LIN {X 0,Y 207.19,Z 445.671,A -85,B 0,C 180,E1 -21067.798,E2 -21067.798} C_VEL
LIN {X 0,Y 206.976,Z 445.696,A -85,B 0,C 180,E1 -21071.756,E2 -21071.756} C_VEL
LIN {X 0,Y 206.869,Z 445.715,A -85,B 0,C 180,E1 -21075.771,E2 -21075.771} C_VEL
LIN {X 0,Y 206.785,Z 445.706,A -85,B 0,C 180,E1 -21079.869,E2 -21079.869} C_VEL
LIN {X 0,Y 206.765,Z 445.704,A -85,B 0,C 180,E1 -21084.072,E2 -21084.072} C_VEL
LIN {X 0,Y 206.745,Z 445.731,A -85,B 0,C 180,E1 -21088.419,E2 -21088.419} C_VEL
LIN {X 0,Y 206.71,Z 445.707,A -85,B 0,C 180,E1 -21092.956,E2 -21092.956} C_VEL
LIN {X 0,Y 206.723,Z 445.722,A -85,B 0,C 180,E1 -21095.321,E2 -21095.321} C_VEL
LIN {X 0,Y 206.668,Z 445.735,A -85,B 0,C 180,E1 -21100.25,E2 -21100.25} C_VEL
LIN {X 0,Y 206.636,Z 445.739,A -85,B 0,C 180,E1 -21105.582,E2 -21105.582} C_VEL
LIN {X 0,Y 206.668,Z 445.737,A -85,B 0,C 180,E1 -21109.751,E2 -21109.751} C_VEL
LIN {X 0,Y 206.733,Z 445.724,A -85,B 0,C 180,E1 -21114.696,E2 -21114.696} C_VEL
LIN {X 0,Y 206.73,Z 445.73,A -85,B 0,C 180,E1 -21119.52,E2 -21119.52} C_VEL
LIN {X 0,Y 207.05,Z 447.125,A -85,B 0,C 180,E1 -21119.722,E2 -21119.722} C_VEL
LIN {X 0,Y 211.426,Z 456.277,A -85,B 0,C 180,E1 -21121.603,E2 -21121.603} C_VEL
LIN {X 0,Y 214.653,Z 464.205,A -85,B 0,C 180,E1 -21123.308,E2 -21123.308} C_VEL
LIN {X 0,Y 217.835,Z 474.221,A -85,B 0,C 180,E1 -21125.577,E2 -21125.577} C_VEL
LIN {X 0,Y 220.061,Z 483.327,A -85,B 0,C 180,E1 -21127.846,E2 -21127.846} C_VEL
LIN {X 0,Y 218.248,Z 491.893,A -85,B 0,C 180,E1 -21129.747,E2 -21129.747} C_VEL
LIN {X 0,Y 215.992,Z 500.319,A -85,B 0,C 180,E1 -21131.995,E2 -21131.995} C_VEL
LIN {X 0,Y 213.676,Z 508.48,A -85,B 0,C 180,E1 -21134.745,E2 -21134.745} C_VEL
LIN {X 0,Y 211.802,Z 515.035,A -85,B 0,C 180,E1 -21137.545,E2 -21137.545} C_VEL
LIN {X 0,Y 210.29,Z 520.267,A -85,B 0,C 180,E1 -21140.381,E2 -21140.381} C_VEL
LIN {X 0,Y 209.024,Z 524.37,A -85,B 0,C 180,E1 -21143.242,E2 -21143.242} C_VEL
LIN {X 0,Y 207.997,Z 527.462,A -85,B 0,C 180,E1 -21146.126,E2 -21146.126} C_VEL
LIN {X 0,Y 207.633,Z 528.989,A -85,B 0,C 180,E1 -21148.061,E2 -21148.061} C_VEL
LIN {X 0,Y 207.465,Z 530.098,A -85,B 0,C 180,E1 -21150,E2 -21150} C_VEL
LIN {X 0,Y 207.463,Z 530.79,A -85,B 0,C 180,E1 -21151.942,E2 -21151.942} C_VEL
LIN {X 0,Y 207.447,Z 531.134,A -85,B 0,C 180,E1 -21155.834,E2 -21155.834} C_VEL
LIN {X 0,Y 207.905,Z 530.696,A -85,B 0,C 180,E1 -21157.772,E2 -21157.772} C_VEL
LIN {X 0,Y 209.475,Z 528.577,A -85,B 0,C 180,E1 -21161.614,E2 -21161.614} C_VEL
LIN {X 0,Y 211.112,Z 525.293,A -85,B 0,C 180,E1 -21165.109,E2 -21165.109} C_VEL
LIN {X 0,Y 212.98,Z 520.951,A -85,B 0,C 180,E1 -21168.27,E2 -21168.27} C_VEL
LIN {X 0,Y 215.03,Z 515.843,A -85,B 0,C 180,E1 -21171.071,E2 -21171.071} C_VEL
LIN {X 0,Y 217.394,Z 509.41,A -85,B 0,C 180,E1 -21173.836,E2 -21173.836} C_VEL
LIN {X 0,Y 220.287,Z 501.361,A -85,B 0,C 180,E1 -21176.53,E2 -21176.53} C_VEL
LIN {X 0,Y 222.893,Z 493.095,A -85,B 0,C 180,E1 -21178.741,E2 -21178.741} C_VEL
LIN {X 0,Y 223.378,Z 491.199,A -85,B 0,C 180,E1 -21179.188,E2 -21179.188} C_VEL
LIN {X 0,Y 223.029,Z 487.399,A -85,B 0,C 180,E1 -21180.278,E2 -21180.278} C_VEL
LIN {X 0,Y 220.921,Z 478.734,A -85,B 0,C 180,E1 -21182.739,E2 -21182.739} C_VEL
LIN {X 0,Y 217.615,Z 468.861,A -85,B 0,C 180,E1 -21185.368,E2 -21185.368} C_VEL
LIN {X 0,Y 213.924,Z 460.069,A -85,B 0,C 180,E1 -21187.6,E2 -21187.6} C_VEL
LIN {X 0,Y 210.239,Z 452.835,A -85,B 0,C 180,E1 -21189.431,E2 -21189.431} C_VEL
LIN {X 0,Y 208.72,Z 449.857,A -85,B 0,C 180,E1 -21190.156,E2 -21190.156} C_VEL
LIN {X 0,Y 207.001,Z 447.117,A -85,B 0,C 180,E1 -21190.871,E2 -21190.871} C_VEL
LIN {X 0,Y 206.686,Z 445.74,A -85,B 0,C 180,E1 -21191.119,E2 -21191.119} C_VEL
LIN {X 0,Y 206.638,Z 445.745,A -85,B 0,C 180,E1 -21195.581,E2 -21195.581} C_VEL
LIN {X 0,Y 206.67,Z 445.738,A -85,B 0,C 180,E1 -21199.75,E2 -21199.75} C_VEL
LIN {X 0,Y 206.735,Z 445.729,A -85,B 0,C 180,E1 -21204.695,E2 -21204.695} C_VEL
LIN {X 0,Y 206.728,Z 445.732,A -85,B 0,C 180,E1 -21209.339,E2 -21209.339} C_VEL
LIN {X 0,Y 206.735,Z 445.734,A -85,B 0,C 180,E1 -21213.772,E2 -21213.772} C_VEL
LIN {X 0,Y 206.86,Z 445.715,A -85,B 0,C 180,E1 -21219.1,E2 -21219.1} C_VEL
LIN {X 0,Y 206.941,Z 445.761,A -85,B 0,C 180,E1 -21219.693,E2 -21219.693} C_VEL
LIN {X 0,Y 209.859,Z 459.288,A -85,B 0,C 180,E1 -21221.594,E2 -21221.594} C_VEL
LIN {X 0,Y 210.707,Z 463.779,A -85,B 0,C 180,E1 -21222.316,E2 -21222.316} C_VEL
LIN {X 0,Y 209.71,Z 475.714,A -85,B 0,C 180,E1 -21224.448,E2 -21224.448} C_VEL
LIN {X 0,Y 208.543,Z 487.804,A -85,B 0,C 180,E1 -21227.099,E2 -21227.099} C_VEL
LIN {X 0,Y 207.569,Z 498.303,A -85,B 0,C 180,E1 -21229.914,E2 -21229.914} C_VEL
LIN {X 0,Y 206.894,Z 506.907,A -85,B 0,C 180,E1 -21232.681,E2 -21232.681} C_VEL
LIN {X 0,Y 206.491,Z 514.452,A -85,B 0,C 180,E1 -21235.608,E2 -21235.608} C_VEL
LIN {X 0,Y 206.658,Z 521.636,A -85,B 0,C 180,E1 -21239.025,E2 -21239.025} C_VEL
LIN {X 0,Y 207.102,Z 526.662,A -85,B 0,C 180,E1 -21241.944,E2 -21241.944} C_VEL
LIN {X 0,Y 208.248,Z 531.871,A -85,B 0,C 180,E1 -21245.811,E2 -21245.811} C_VEL
LIN {X 0,Y 210.256,Z 535.477,A -85,B 0,C 180,E1 -21249.621,E2 -21249.621} C_VEL
LIN {X 0,Y 213.286,Z 537.641,A -85,B 0,C 180,E1 -21253.336,E2 -21253.336} C_VEL
LIN {X 0,Y 216.951,Z 538.342,A -85,B 0,C 180,E1 -21256.951,E2 -21256.951} C_VEL
LIN {X 0,Y 221.52,Z 537.675,A -85,B 0,C 180,E1 -21260.425,E2 -21260.425} C_VEL
LIN {X 0,Y 226.914,Z 535.59,A -85,B 0,C 180,E1 -21263.743,E2 -21263.743} C_VEL
LIN {X 0,Y 233.04,Z 532.075,A -85,B 0,C 180,E1 -21266.896,E2 -21266.896} C_VEL
LIN {X 0,Y 239.903,Z 527.051,A -85,B 0,C 180,E1 -21269.869,E2 -21269.869} C_VEL
LIN {X 0,Y 247.431,Z 520.392,A -85,B 0,C 180,E1 -21272.661,E2 -21272.661} C_VEL
LIN {X 0,Y 248.551,Z 519.043,A -85,B 0,C 180,E1 -21273.462,E2 -21273.462} C_VEL
LIN {X 0,Y 249.773,Z 517.18,A -85,B 0,C 180,E1 -21275.314,E2 -21275.314} C_VEL
LIN {X 0,Y 250.027,Z 516.636,A -85,B 0,C 180,E1 -21276.177,E2 -21276.177} C_VEL
LIN {X 0,Y 250.154,Z 516.146,A -85,B 0,C 180,E1 -21278.176,E2 -21278.176} C_VEL
LIN {X 0,Y 249.645,Z 516.912,A -85,B 0,C 180,E1 -21280.526,E2 -21280.526} C_VEL
LIN {X 0,Y 248.76,Z 518.828,A -85,B 0,C 180,E1 -21282.73,E2 -21282.73} C_VEL
LIN {X 0,Y 248.092,Z 520.223,A -85,B 0,C 180,E1 -21283.715,E2 -21283.715} C_VEL
LIN {X 0,Y 247.046,Z 522.094,A -85,B 0,C 180,E1 -21284.666,E2 -21284.666} C_VEL
LIN {X 0,Y 243.621,Z 527.852,A -85,B 0,C 180,E1 -21286.954,E2 -21286.954} C_VEL
LIN {X 0,Y 238.302,Z 537.311,A -85,B 0,C 180,E1 -21290.471,E2 -21290.471} C_VEL
LIN {X 0,Y 232.802,Z 546.857,A -85,B 0,C 180,E1 -21293.936,E2 -21293.936} C_VEL
LIN {X 0,Y 227.947,Z 554.484,A -85,B 0,C 180,E1 -21296.82,E2 -21296.82} C_VEL
LIN {X 0,Y 221.36,Z 563.244,A -85,B 0,C 180,E1 -21300.52,E2 -21300.52} C_VEL
LIN {X 0,Y 216.239,Z 569.715,A -85,B 0,C 180,E1 -21303.974,E2 -21303.974} C_VEL
LIN {X 0,Y 212.413,Z 573.997,A -85,B 0,C 180,E1 -21306.876,E2 -21306.876} C_VEL
LIN {X 0,Y 210.69,Z 575.213,A -85,B 0,C 180,E1 -21307.802,E2 -21307.802} C_VEL
LIN {X 0,Y 206.361,Z 576.777,A -85,B 0,C 180,E1 -21309.173,E2 -21309.173} C_VEL
LIN {X 0,Y 202.257,Z 578.001,A -85,B 0,C 180,E1 -21310.633,E2 -21310.633} C_VEL
LIN {X 0,Y 200.915,Z 578.675,A -85,B 0,C 180,E1 -21311.677,E2 -21311.677} C_VEL
LIN {X 0,Y 199.246,Z 580.859,A -85,B 0,C 180,E1 -21315.705,E2 -21315.705} C_VEL
LIN {X 0,Y 198.485,Z 584.504,A -85,B 0,C 180,E1 -21318.77,E2 -21318.77} C_VEL
LIN {X 0,Y 198.527,Z 587.544,A -85,B 0,C 180,E1 -21322.401,E2 -21322.401} C_VEL
LIN {X 0,Y 199.087,Z 589.273,A -85,B 0,C 180,E1 -21325.951,E2 -21325.951} C_VEL
LIN {X 0,Y 200.122,Z 589.738,A -85,B 0,C 180,E1 -21330,E2 -21330} C_VEL
LIN {X 0,Y 199.15,Z 588.129,A -85,B 0,C 180,E1 -21334.047,E2 -21334.047} C_VEL
LIN {X 0,Y 198.609,Z 585.183,A -85,B 0,C 180,E1 -21337.773,E2 -21337.773} C_VEL
LIN {X 0,Y 198.547,Z 581.133,A -85,B 0,C 180,E1 -21341.226,E2 -21341.226} C_VEL
LIN {X 0,Y 199.107,Z 576.342,A -85,B 0,C 180,E1 -21344.305,E2 -21344.305} C_VEL
LIN {X 0,Y 200.206,Z 570.306,A -85,B 0,C 180,E1 -21347.36,E2 -21347.36} C_VEL
LIN {X 0,Y 202.241,Z 562.871,A -85,B 0,C 180,E1 -21350.334,E2 -21350.334} C_VEL
LIN {X 0,Y 203.98,Z 555.277,A -85,B 0,C 180,E1 -21352.806,E2 -21352.806} C_VEL
LIN {X 0,Y 205.4,Z 544.939,A -85,B 0,C 180,E1 -21355.593,E2 -21355.593} C_VEL
LIN {X 0,Y 206.435,Z 534.473,A -85,B 0,C 180,E1 -21357.897,E2 -21357.897} C_VEL
LIN {X 0,Y 206.989,Z 522.611,A -85,B 0,C 180,E1 -21360.053,E2 -21360.053} C_VEL
LIN {X 0,Y 206.838,Z 510.847,A -85,B 0,C 180,E1 -21361.847,E2 -21361.847} C_VEL
LIN {X 0,Y 205.857,Z 498.168,A -85,B 0,C 180,E1 -21363.484,E2 -21363.484} C_VEL
LIN {X 0,Y 203.822,Z 484.285,A -85,B 0,C 180,E1 -21364.972,E2 -21364.972} C_VEL
LIN {X 0,Y 202.372,Z 476.893,A -85,B 0,C 180,E1 -21365.66,E2 -21365.66} C_VEL
LIN {X 0,Y 203.976,Z 470.853,A -85,B 0,C 180,E1 -21369.526,E2 -21369.526} C_VEL
LIN {X 0,Y 203.993,Z 468.815,A -85,B 0,C 180,E1 -21370.888,E2 -21370.888} C_VEL
LIN {X 0,Y 202.951,Z 463.172,A -85,B 0,C 180,E1 -21374.924,E2 -21374.924} C_VEL
LIN {X 0,Y 201.676,Z 456.469,A -85,B 0,C 180,E1 -21380.054,E2 -21380.054} C_VEL
LIN {X 0,Y 200.597,Z 450.842,A -85,B 0,C 180,E1 -21384.723,E2 -21384.723} C_VEL
LIN {X 0,Y 199.668,Z 446.619,A -85,B 0,C 180,E1 -21388.723,E2 -21388.723} C_VEL
LIN {X 0,Y 199.686,Z 446.608,A -85,B 0,C 180,E1 -21392.772,E2 -21392.772} C_VEL
LIN {X 0,Y 199.75,Z 446.605,A -85,B 0,C 180,E1 -21397.231,E2 -21397.231} C_VEL
LIN {X 0,Y 199.838,Z 446.597,A -85,B 0,C 180,E1 -21401.722,E2 -21401.722} C_VEL
LIN {X 0,Y 199.837,Z 446.596,A -85,B 0,C 180,E1 -21405.749,E2 -21405.749} C_VEL
LIN {X 0,Y 200.023,Z 446.571,A -85,B 0,C 180,E1 -21409.882,E2 -21409.882} C_VEL
LIN {X 0,Y 200.023,Z 446.572,A -85,B 0,C 180,E1 -21413.95,E2 -21413.95} C_VEL
LIN {X 0,Y 200.323,Z 446.531,A -85,B 0,C 180,E1 -21417.99,E2 -21417.99} C_VEL
LIN {X 0,Y 200.484,Z 446.513,A -85,B 0,C 180,E1 -21420,E2 -21420} C_VEL
LIN {X 0,Y 200.034,Z 446.566,A -85,B 0,C 180,E1 -21424.03,E2 -21424.03} C_VEL
LIN {X 0,Y 200.133,Z 446.551,A -85,B 0,C 180,E1 -21428.075,E2 -21428.075} C_VEL
LIN {X 0,Y 199.907,Z 446.573,A -85,B 0,C 180,E1 -21432.178,E2 -21432.178} C_VEL
LIN {X 0,Y 199.806,Z 446.595,A -85,B 0,C 180,E1 -21436.344,E2 -21436.344} C_VEL
LIN {X 0,Y 199.701,Z 446.581,A -85,B 0,C 180,E1 -21440.606,E2 -21440.606} C_VEL
LIN {X 0,Y 199.674,Z 446.596,A -85,B 0,C 180,E1 -21444.985,E2 -21444.985} C_VEL
LIN {X 0,Y 199.676,Z 446.609,A -85,B 0,C 180,E1 -21449.523,E2 -21449.523} C_VEL
LIN {X 0,Y 199.665,Z 446.586,A -85,B 0,C 180,E1 -21452.353,E2 -21452.353} C_VEL
LIN {X 0,Y 199.641,Z 446.615,A -85,B 0,C 180,E1 -21456.76,E2 -21456.76} C_VEL
LIN {X 0,Y 199.64,Z 446.614,A -85,B 0,C 180,E1 -21459.321,E2 -21459.321} C_VEL
LIN {X 0,Y 199.582,Z 446.615,A -85,B 0,C 180,E1 -21464.771,E2 -21464.771} C_VEL
LIN {X 0,Y 199.584,Z 446.615,A -85,B 0,C 180,E1 -21468.006,E2 -21468.006} C_VEL
LIN {X 0,Y 199.643,Z 446.61,A -85,B 0,C 180,E1 -21470.757,E2 -21470.757} C_VEL
LIN {X 0,Y 199.637,Z 446.611,A -85,B 0,C 180,E1 -21475.719,E2 -21475.719} C_VEL
LIN {X 0,Y 199.709,Z 446.618,A -85,B 0,C 180,E1 -21478.222,E2 -21478.222} C_VEL
LIN {X 0,Y 200.279,Z 448.714,A -85,B 0,C 180,E1 -21478.553,E2 -21478.553} C_VEL
LIN {X 0,Y 203.236,Z 454.419,A -85,B 0,C 180,E1 -21479.828,E2 -21479.828} C_VEL
LIN {X 0,Y 207.197,Z 463.513,A -85,B 0,C 180,E1 -21481.874,E2 -21481.874} C_VEL
LIN {X 0,Y 210.647,Z 473.754,A -85,B 0,C 180,E1 -21484.296,E2 -21484.296} C_VEL
LIN {X 0,Y 213.055,Z 483.02,A -85,B 0,C 180,E1 -21486.682,E2 -21486.682} C_VEL
LIN {X 0,Y 213.458,Z 484.98,A -85,B 0,C 180,E1 -21487.205,E2 -21487.205} C_VEL
LIN {X 0,Y 212.605,Z 489.566,A -85,B 0,C 180,E1 -21488.241,E2 -21488.241} C_VEL
LIN {X 0,Y 210.214,Z 498.336,A -85,B 0,C 180,E1 -21490.469,E2 -21490.469} C_VEL
LIN {X 0,Y 207.744,Z 507.098,A -85,B 0,C 180,E1 -21493.289,E2 -21493.289} C_VEL
LIN {X 0,Y 205.515,Z 514.171,A -85,B 0,C 180,E1 -21496.151,E2 -21496.151} C_VEL
LIN {X 0,Y 203.909,Z 519.784,A -85,B 0,C 180,E1 -21499.073,E2 -21499.073} C_VEL
LIN {X 0,Y 202.407,Z 524.24,A -85,B 0,C 180,E1 -21502.017,E2 -21502.017} C_VEL
LIN {X 0,Y 201.594,Z 526.596,A -85,B 0,C 180,E1 -21503.997,E2 -21503.997} C_VEL
LIN {X 0,Y 200.614,Z 530.042,A -85,B 0,C 180,E1 -21507.993,E2 -21507.993} C_VEL
LIN {X 0,Y 200.439,Z 531.132,A -85,B 0,C 180,E1 -21510,E2 -21510} C_VEL
LIN {X 0,Y 200.439,Z 531.816,A -85,B 0,C 180,E1 -21512.01,E2 -21512.01} C_VEL
LIN {X 0,Y 200.45,Z 532.142,A -85,B 0,C 180,E1 -21516.038,E2 -21516.038} C_VEL
LIN {X 0,Y 200.938,Z 531.686,A -85,B 0,C 180,E1 -21518.043,E2 -21518.043} C_VEL
LIN {X 0,Y 202.594,Z 529.548,A -85,B 0,C 180,E1 -21522.014,E2 -21522.014} C_VEL
LIN {X 0,Y 204.334,Z 526.242,A -85,B 0,C 180,E1 -21525.621,E2 -21525.621} C_VEL
LIN {X 0,Y 206.309,Z 521.872,A -85,B 0,C 180,E1 -21528.883,E2 -21528.883} C_VEL
LIN {X 0,Y 208.478,Z 516.742,A -85,B 0,C 180,E1 -21531.767,E2 -21531.767} C_VEL
LIN {X 0,Y 210.97,Z 510.284,A -85,B 0,C 180,E1 -21534.609,E2 -21534.609} C_VEL
LIN {X 0,Y 214.022,Z 502.204,A -85,B 0,C 180,E1 -21537.37,E2 -21537.37} C_VEL
LIN {X 0,Y 216.73,Z 493.898,A -85,B 0,C 180,E1 -21539.639,E2 -21539.639} C_VEL
LIN {X 0,Y 216.981,Z 492.026,A -85,B 0,C 180,E1 -21540.136,E2 -21540.136} C_VEL
LIN {X 0,Y 215.523,Z 484.475,A -85,B 0,C 180,E1 -21542.46,E2 -21542.46} C_VEL
LIN {X 0,Y 213.086,Z 476.2,A -85,B 0,C 180,E1 -21544.877,E2 -21544.877} C_VEL
LIN {X 0,Y 209.542,Z 466.453,A -85,B 0,C 180,E1 -21547.55,E2 -21547.55} C_VEL
LIN {X 0,Y 205.754,Z 458.208,A -85,B 0,C 180,E1 -21549.776,E2 -21549.776} C_VEL
LIN {X 0,Y 201.012,Z 450.086,A -85,B 0,C 180,E1 -21552.073,E2 -21552.073} C_VEL
LIN {X 0,Y 199.757,Z 447.503,A -85,B 0,C 180,E1 -21552.701,E2 -21552.701} C_VEL
LIN {X 0,Y 199.609,Z 446.62,A -85,B 0,C 180,E1 -21552.905,E2 -21552.905} C_VEL
LIN {X 0,Y 199.586,Z 446.619,A -85,B 0,C 180,E1 -21558.006,E2 -21558.006} C_VEL
LIN {X 0,Y 199.645,Z 446.61,A -85,B 0,C 180,E1 -21560.757,E2 -21560.757} C_VEL
LIN {X 0,Y 199.639,Z 446.616,A -85,B 0,C 180,E1 -21565.718,E2 -21565.718} C_VEL
LIN {X 0,Y 199.708,Z 446.603,A -85,B 0,C 180,E1 -21568.138,E2 -21568.138} C_VEL
LIN {X 0,Y 199.69,Z 446.609,A -85,B 0,C 180,E1 -21572.772,E2 -21572.772} C_VEL
LIN {X 0,Y 199.732,Z 446.604,A -85,B 0,C 180,E1 -21577.228,E2 -21577.228} C_VEL
LIN {X 0,Y 199.853,Z 446.586,A -85,B 0,C 180,E1 -21579.604,E2 -21579.604} C_VEL
LIN {X 0,Y 202.93,Z 460.743,A -85,B 0,C 180,E1 -21581.68,E2 -21581.68} C_VEL
LIN {X 0,Y 203.546,Z 463.603,A -85,B 0,C 180,E1 -21582.155,E2 -21582.155} C_VEL
LIN {X 0,Y 202.597,Z 475.994,A -85,B 0,C 180,E1 -21584.404,E2 -21584.404} C_VEL
LIN {X 0,Y 201.416,Z 488.221,A -85,B 0,C 180,E1 -21587.147,E2 -21587.147} C_VEL
LIN {X 0,Y 200.483,Z 498.323,A -85,B 0,C 180,E1 -21589.905,E2 -21589.905} C_VEL
LIN {X 0,Y 199.739,Z 507.428,A -85,B 0,C 180,E1 -21592.926,E2 -21592.926} C_VEL
LIN {X 0,Y 199.4,Z 516.244,A -85,B 0,C 180,E1 -21596.463,E2 -21596.463} C_VEL
LIN {X 0,Y 199.701,Z 523.362,A -85,B 0,C 180,E1 -21600,E2 -21600} C_VEL
LIN {X 0,Y 200.319,Z 528.269,A -85,B 0,C 180,E1 -21603.016,E2 -21603.016} C_VEL
LIN {X 0,Y 201.657,Z 533.42,A -85,B 0,C 180,E1 -21607.006,E2 -21607.006} C_VEL
LIN {X 0,Y 203.32,Z 536.262,A -85,B 0,C 180,E1 -21609.952,E2 -21609.952} C_VEL
LIN {X 0,Y 206.48,Z 538.715,A -85,B 0,C 180,E1 -21613.784,E2 -21613.784} C_VEL
LIN {X 0,Y 210.331,Z 539.813,A -85,B 0,C 180,E1 -21617.501,E2 -21617.501} C_VEL
LIN {X 0,Y 215.126,Z 539.487,A -85,B 0,C 180,E1 -21621.061,E2 -21621.061} C_VEL
LIN {X 0,Y 220.747,Z 537.81,A -85,B 0,C 180,E1 -21624.449,E2 -21624.449} C_VEL
LIN {X 0,Y 227.18,Z 534.742,A -85,B 0,C 180,E1 -21627.648,E2 -21627.648} C_VEL
LIN {X 0,Y 234.321,Z 530.175,A -85,B 0,C 180,E1 -21630.656,E2 -21630.656} C_VEL
LIN {X 0,Y 240.103,Z 525.747,A -85,B 0,C 180,E1 -21632.786,E2 -21632.786} C_VEL
LIN {X 0,Y 242.117,Z 524.055,A -85,B 0,C 180,E1 -21633.471,E2 -21633.471} C_VEL
LIN {X 0,Y 243.447,Z 522.835,A -85,B 0,C 180,E1 -21634.259,E2 -21634.259} C_VEL
LIN {X 0,Y 244.111,Z 522.024,A -85,B 0,C 180,E1 -21635.156,E2 -21635.156} C_VEL
LIN {X 0,Y 244.733,Z 521.284,A -85,B 0,C 180,E1 -21636.478,E2 -21636.478} C_VEL
LIN {X 0,Y 244.703,Z 521.333,A -85,B 0,C 180,E1 -21639.187,E2 -21639.187} C_VEL
LIN {X 0,Y 243.992,Z 522.763,A -85,B 0,C 180,E1 -21641.503,E2 -21641.503} C_VEL
LIN {X 0,Y 243.477,Z 523.818,A -85,B 0,C 180,E1 -21642.567,E2 -21642.567} C_VEL
LIN {X 0,Y 242.516,Z 525.419,A -85,B 0,C 180,E1 -21643.573,E2 -21643.573} C_VEL
LIN {X 0,Y 239.087,Z 530.446,A -85,B 0,C 180,E1 -21645.788,E2 -21645.788} C_VEL
LIN {X 0,Y 233.115,Z 539.533,A -85,B 0,C 180,E1 -21649.41,E2 -21649.41} C_VEL
LIN {X 0,Y 227.223,Z 548.426,A -85,B 0,C 180,E1 -21652.905,E2 -21652.905} C_VEL
LIN {X 0,Y 222.878,Z 554.552,A -85,B 0,C 180,E1 -21655.417,E2 -21655.417} C_VEL
LIN {X 0,Y 215.2,Z 563.657,A -85,B 0,C 180,E1 -21659.588,E2 -21659.588} C_VEL
LIN {X 0,Y 209.881,Z 569.651,A -85,B 0,C 180,E1 -21663.124,E2 -21663.124} C_VEL
LIN {X 0,Y 205.087,Z 574.433,A -85,B 0,C 180,E1 -21666.79,E2 -21666.79} C_VEL
LIN {X 0,Y 202.264,Z 577.242,A -85,B 0,C 180,E1 -21669.745,E2 -21669.745} C_VEL
LIN {X 0,Y 200.915,Z 578.675,A -85,B 0,C 180,E1 -21671.677,E2 -21671.677} C_VEL
LIN {X 0,Y 199.435,Z 579.718,A -85,B 0,C 180,E1 -21673.286,E2 -21673.286} C_VEL
LIN {X 0,Y 195.566,Z 581.659,A -85,B 0,C 180,E1 -21675.873,E2 -21675.873} C_VEL
LIN {X 0,Y 192.65,Z 583.358,A -85,B 0,C 180,E1 -21677.997,E2 -21677.997} C_VEL
LIN {X 0,Y 191.433,Z 584.744,A -85,B 0,C 180,E1 -21679.676,E2 -21679.676} C_VEL
LIN {X 0,Y 191.333,Z 585.156,A -85,B 0,C 180,E1 -21680.249,E2 -21680.249} C_VEL
LIN {X 0,Y 191.592,Z 587.423,A -85,B 0,C 180,E1 -21683.682,E2 -21683.682} C_VEL
LIN {X 0,Y 191.997,Z 588.26,A -85,B 0,C 180,E1 -21685.801,E2 -21685.801} C_VEL
LIN {X 0,Y 193.054,Z 588.714,A -85,B 0,C 180,E1 -21690,E2 -21690} C_VEL
LIN {X 0,Y 192.059,Z 587.078,A -85,B 0,C 180,E1 -21694.197,E2 -21694.197} C_VEL
LIN {X 0,Y 191.535,Z 584.332,A -85,B 0,C 180,E1 -21697.816,E2 -21697.816} C_VEL
LIN {X 0,Y 191.534,Z 580.037,A -85,B 0,C 180,E1 -21701.643,E2 -21701.643} C_VEL
LIN {X 0,Y 192.156,Z 575.223,A -85,B 0,C 180,E1 -21704.834,E2 -21704.834} C_VEL
LIN {X 0,Y 193.386,Z 569.164,A -85,B 0,C 180,E1 -21707.993,E2 -21707.993} C_VEL
LIN {X 0,Y 195.54,Z 561.705,A -85,B 0,C 180,E1 -21711.064,E2 -21711.064} C_VEL
LIN {X 0,Y 196.97,Z 555.75,A -85,B 0,C 180,E1 -21713.109,E2 -21713.109} C_VEL
LIN {X 0,Y 198.491,Z 545.717,A -85,B 0,C 180,E1 -21715.986,E2 -21715.986} C_VEL
LIN {X 0,Y 199.607,Z 535.813,A -85,B 0,C 180,E1 -21718.33,E2 -21718.33} C_VEL
LIN {X 0,Y 200.372,Z 524.472,A -85,B 0,C 180,E1 -21720.569,E2 -21720.569} C_VEL
LIN {X 0,Y 200.422,Z 512.996,A -85,B 0,C 180,E1 -21722.472,E2 -21722.472} C_VEL
LIN {X 0,Y 199.621,Z 500.032,A -85,B 0,C 180,E1 -21724.284,E2 -21724.284} C_VEL
LIN {X 0,Y 197.898,Z 486.713,A -85,B 0,C 180,E1 -21725.864,E2 -21725.864} C_VEL
LIN {X 0,Y 195.802,Z 475.799,A -85,B 0,C 180,E1 -21726.993,E2 -21726.993} C_VEL
LIN {X 0,Y 196.961,Z 471.336,A -85,B 0,C 180,E1 -21729.961,E2 -21729.961} C_VEL
LIN {X 0,Y 196.874,Z 469.24,A -85,B 0,C 180,E1 -21731.439,E2 -21731.439} C_VEL
LIN {X 0,Y 195.746,Z 463.258,A -85,B 0,C 180,E1 -21735.895,E2 -21735.895} C_VEL
LIN {X 0,Y 194.602,Z 457.171,A -85,B 0,C 180,E1 -21740.802,E2 -21740.802} C_VEL
LIN {X 0,Y 193.789,Z 452.856,A -85,B 0,C 180,E1 -21744.531,E2 -21744.531} C_VEL
LIN {X 0,Y 192.628,Z 447.491,A -85,B 0,C 180,E1 -21749.667,E2 -21749.667} C_VEL
LIN {X 0,Y 192.599,Z 447.495,A -85,B 0,C 180,E1 -21754.031,E2 -21754.031} C_VEL
LIN {X 0,Y 192.712,Z 447.482,A -85,B 0,C 180,E1 -21756.35,E2 -21756.35} C_VEL
LIN {X 0,Y 192.782,Z 447.475,A -85,B 0,C 180,E1 -21761.413,E2 -21761.413} C_VEL
LIN {X 0,Y 192.765,Z 447.475,A -85,B 0,C 180,E1 -21765.214,E2 -21765.214} C_VEL
LIN {X 0,Y 192.945,Z 447.453,A -85,B 0,C 180,E1 -21769.567,E2 -21769.567} C_VEL
LIN {X 0,Y 192.985,Z 447.447,A -85,B 0,C 180,E1 -21773.728,E2 -21773.728} C_VEL
LIN {X 0,Y 193.265,Z 447.411,A -85,B 0,C 180,E1 -21777.916,E2 -21777.916} C_VEL
LIN {X 0,Y 193.447,Z 447.389,A -85,B 0,C 180,E1 -21780,E2 -21780} C_VEL
LIN {X 0,Y 192.981,Z 447.443,A -85,B 0,C 180,E1 -21784.177,E2 -21784.177} C_VEL
LIN {X 0,Y 193.08,Z 447.432,A -85,B 0,C 180,E1 -21788.372,E2 -21788.372} C_VEL
LIN {X 0,Y 193.011,Z 447.44,A -85,B 0,C 180,E1 -21790.539,E2 -21790.539} C_VEL
LIN {X 0,Y 192.759,Z 447.471,A -85,B 0,C 180,E1 -21796.959,E2 -21796.959} C_VEL
LIN {X 0,Y 192.637,Z 447.451,A -85,B 0,C 180,E1 -21801.398,E2 -21801.398} C_VEL
LIN {X 0,Y 192.665,Z 447.458,A -85,B 0,C 180,E1 -21804.225,E2 -21804.225} C_VEL
LIN {X 0,Y 192.651,Z 447.485,A -85,B 0,C 180,E1 -21808.893,E2 -21808.893} C_VEL
LIN {X 0,Y 192.601,Z 447.462,A -85,B 0,C 180,E1 -21813.186,E2 -21813.186} C_VEL
LIN {X 0,Y 192.611,Z 447.489,A -85,B 0,C 180,E1 -21816.608,E2 -21816.608} C_VEL
LIN {X 0,Y 192.525,Z 447.498,A -85,B 0,C 180,E1 -21821.078,E2 -21821.078} C_VEL
LIN {X 0,Y 192.515,Z 447.501,A -85,B 0,C 180,E1 -21826.083,E2 -21826.083} C_VEL
LIN {X 0,Y 192.543,Z 447.496,A -85,B 0,C 180,E1 -21830.043,E2 -21830.043} C_VEL
LIN {X 0,Y 192.6,Z 447.485,A -85,B 0,C 180,E1 -21834.279,E2 -21834.279} C_VEL
LIN {X 0,Y 192.599,Z 447.49,A -85,B 0,C 180,E1 -21836.776,E2 -21836.776} C_VEL
LIN {X 0,Y 193.353,Z 449.848,A -85,B 0,C 180,E1 -21837.199,E2 -21837.199} C_VEL
LIN {X 0,Y 194.46,Z 451.537,A -85,B 0,C 180,E1 -21837.652,E2 -21837.652} C_VEL
LIN {X 0,Y 199.494,Z 462.43,A -85,B 0,C 180,E1 -21840.226,E2 -21840.226} C_VEL
LIN {X 0,Y 202.868,Z 471.467,A -85,B 0,C 180,E1 -21842.453,E2 -21842.453} C_VEL
LIN {X 0,Y 205.528,Z 480.807,A -85,B 0,C 180,E1 -21844.891,E2 -21844.891} C_VEL
LIN {X 0,Y 206.856,Z 486.679,A -85,B 0,C 180,E1 -21846.541,E2 -21846.541} C_VEL
LIN {X 0,Y 206.465,Z 489.443,A -85,B 0,C 180,E1 -21847.208,E2 -21847.208} C_VEL
LIN {X 0,Y 204.12,Z 497.874,A -85,B 0,C 180,E1 -21849.335,E2 -21849.335} C_VEL
LIN {X 0,Y 201.817,Z 505.592,A -85,B 0,C 180,E1 -21851.735,E2 -21851.735} C_VEL
LIN {X 0,Y 199.46,Z 513.12,A -85,B 0,C 180,E1 -21854.677,E2 -21854.677} C_VEL
LIN {X 0,Y 197.578,Z 519.14,A -85,B 0,C 180,E1 -21857.677,E2 -21857.677} C_VEL
LIN {X 0,Y 195.96,Z 523.94,A -85,B 0,C 180,E1 -21860.713,E2 -21860.713} C_VEL
LIN {X 0,Y 194.611,Z 527.667,A -85,B 0,C 180,E1 -21863.781,E2 -21863.781} C_VEL
LIN {X 0,Y 193.594,Z 531.094,A -85,B 0,C 180,E1 -21867.92,E2 -21867.92} C_VEL
LIN {X 0,Y 193.412,Z 532.166,A -85,B 0,C 180,E1 -21870,E2 -21870} C_VEL
LIN {X 0,Y 193.414,Z 532.841,A -85,B 0,C 180,E1 -21872.083,E2 -21872.083} C_VEL
LIN {X 0,Y 193.457,Z 533.15,A -85,B 0,C 180,E1 -21876.257,E2 -21876.257} C_VEL
LIN {X 0,Y 193.976,Z 532.676,A -85,B 0,C 180,E1 -21878.333,E2 -21878.333} C_VEL
LIN {X 0,Y 195.722,Z 530.52,A -85,B 0,C 180,E1 -21882.442,E2 -21882.442} C_VEL
LIN {X 0,Y 197.507,Z 527.27,A -85,B 0,C 180,E1 -21886.102,E2 -21886.102} C_VEL
LIN {X 0,Y 199.665,Z 522.793,A -85,B 0,C 180,E1 -21889.536,E2 -21889.536} C_VEL
LIN {X 0,Y 201.937,Z 517.644,A -85,B 0,C 180,E1 -21892.51,E2 -21892.51} C_VEL
LIN {X 0,Y 204.586,Z 511.159,A -85,B 0,C 180,E1 -21895.43,E2 -21895.43} C_VEL
LIN {X 0,Y 207.788,Z 503.05,A -85,B 0,C 180,E1 -21898.264,E2 -21898.264} C_VEL
LIN {X 0,Y 210.534,Z 494.73,A -85,B 0,C 180,E1 -21900.596,E2 -21900.596} C_VEL
LIN {X 0,Y 209.71,Z 489.105,A -85,B 0,C 180,E1 -21902.426,E2 -21902.426} C_VEL
LIN {X 0,Y 207.732,Z 481.349,A -85,B 0,C 180,E1 -21904.873,E2 -21904.873} C_VEL
LIN {X 0,Y 204.487,Z 471.626,A -85,B 0,C 180,E1 -21907.768,E2 -21907.768} C_VEL
LIN {X 0,Y 200.656,Z 462.739,A -85,B 0,C 180,E1 -21910.356,E2 -21910.356} C_VEL
LIN {X 0,Y 196.945,Z 455.828,A -85,B 0,C 180,E1 -21912.428,E2 -21912.428} C_VEL
LIN {X 0,Y 194.303,Z 451.363,A -85,B 0,C 180,E1 -21913.784,E2 -21913.784} C_VEL
LIN {X 0,Y 192.862,Z 448.913,A -85,B 0,C 180,E1 -21914.504,E2 -21914.504} C_VEL
LIN {X 0,Y 192.56,Z 447.495,A -85,B 0,C 180,E1 -21914.853,E2 -21914.853} C_VEL
LIN {X 0,Y 192.544,Z 447.496,A -85,B 0,C 180,E1 -21920.043,E2 -21920.043} C_VEL
LIN {X 0,Y 192.602,Z 447.488,A -85,B 0,C 180,E1 -21924.279,E2 -21924.279} C_VEL
LIN {X 0,Y 192.612,Z 447.491,A -85,B 0,C 180,E1 -21929.28,E2 -21929.28} C_VEL
LIN {X 0,Y 192.668,Z 447.48,A -85,B 0,C 180,E1 -21931.692,E2 -21931.692} C_VEL
LIN {X 0,Y 192.69,Z 447.479,A -85,B 0,C 180,E1 -21936.346,E2 -21936.346} C_VEL
LIN {X 0,Y 192.807,Z 447.463,A -85,B 0,C 180,E1 -21939.519,E2 -21939.519} C_VEL
LIN {X 0,Y 195.896,Z 461.787,A -85,B 0,C 180,E1 -21941.704,E2 -21941.704} C_VEL
LIN {X 0,Y 196.488,Z 465.252,A -85,B 0,C 180,E1 -21942.3,E2 -21942.3} C_VEL
LIN {X 0,Y 195.311,Z 477.423,A -85,B 0,C 180,E1 -21944.61,E2 -21944.61} C_VEL
LIN {X 0,Y 194.179,Z 489.47,A -85,B 0,C 180,E1 -21947.457,E2 -21947.457} C_VEL
LIN {X 0,Y 193.363,Z 498.67,A -85,B 0,C 180,E1 -21950.058,E2 -21950.058} C_VEL
LIN {X 0,Y 192.587,Z 507.927,A -85,B 0,C 180,E1 -21953.188,E2 -21953.188} C_VEL
LIN {X 0,Y 192.333,Z 516.879,A -85,B 0,C 180,E1 -21956.858,E2 -21956.858} C_VEL
LIN {X 0,Y 192.615,Z 523.144,A -85,B 0,C 180,E1 -21960,E2 -21960} C_VEL
LIN {X 0,Y 193.251,Z 528.357,A -85,B 0,C 180,E1 -21963.127,E2 -21963.127} C_VEL
LIN {X 0,Y 194.632,Z 533.804,A -85,B 0,C 180,E1 -21967.26,E2 -21967.26} C_VEL
LIN {X 0,Y 196.359,Z 536.893,A -85,B 0,C 180,E1 -21970.309,E2 -21970.309} C_VEL
LIN {X 0,Y 199.685,Z 539.745,A -85,B 0,C 180,E1 -21974.262,E2 -21974.262} C_VEL
LIN {X 0,Y 203.722,Z 541.181,A -85,B 0,C 180,E1 -21978.088,E2 -21978.088} C_VEL
LIN {X 0,Y 208.735,Z 541.246,A -85,B 0,C 180,E1 -21981.738,E2 -21981.738} C_VEL
LIN {X 0,Y 214.617,Z 539.979,A -85,B 0,C 180,E1 -21985.195,E2 -21985.195} C_VEL
LIN {X 0,Y 221.307,Z 537.296,A -85,B 0,C 180,E1 -21988.447,E2 -21988.447} C_VEL
LIN {X 0,Y 228.765,Z 533.26,A -85,B 0,C 180,E1 -21991.484,E2 -21991.484} C_VEL
LIN {X 0,Y 236.857,Z 527.687,A -85,B 0,C 180,E1 -21994.317,E2 -21994.317} C_VEL
LIN {X 0,Y 238.879,Z 526.014,A -85,B 0,C 180,E1 -21996.044,E2 -21996.044} C_VEL
LIN {X 0,Y 239.284,Z 525.714,A -85,B 0,C 180,E1 -21997.531,E2 -21997.531} C_VEL
LIN {X 0,Y 238.845,Z 526.705,A -85,B 0,C 180,E1 -22000.342,E2 -22000.342} C_VEL
LIN {X 0,Y 237.854,Z 528.565,A -85,B 0,C 180,E1 -22002.379,E2 -22002.379} C_VEL
LIN {X 0,Y 235.9,Z 531.152,A -85,B 0,C 180,E1 -22003.761,E2 -22003.761} C_VEL
LIN {X 0,Y 229.224,Z 539.934,A -85,B 0,C 180,E1 -22007.582,E2 -22007.582} C_VEL
LIN {X 0,Y 223.192,Z 547.915,A -85,B 0,C 180,E1 -22010.966,E2 -22010.966} C_VEL
LIN {X 0,Y 217.109,Z 555.525,A -85,B 0,C 180,E1 -22014.36,E2 -22014.36} C_VEL
LIN {X 0,Y 209.11,Z 563.997,A -85,B 0,C 180,E1 -22018.604,E2 -22018.604} C_VEL
LIN {X 0,Y 203.555,Z 569.523,A -85,B 0,C 180,E1 -22022.218,E2 -22022.218} C_VEL
LIN {X 0,Y 199.694,Z 572.928,A -85,B 0,C 180,E1 -22025.018,E2 -22025.018} C_VEL
LIN {X 0,Y 195.381,Z 576.605,A -85,B 0,C 180,E1 -22029.267,E2 -22029.267} C_VEL
LIN {X 0,Y 193.12,Z 578.716,A -85,B 0,C 180,E1 -22033.074,E2 -22033.074} C_VEL
LIN {X 0,Y 192.424,Z 579.555,A -85,B 0,C 180,E1 -22034.916,E2 -22034.916} C_VEL
LIN {X 0,Y 191.485,Z 583.519,A -85,B 0,C 180,E1 -22038.353,E2 -22038.353} C_VEL
LIN {X 0,Y 191.333,Z 585.156,A -85,B 0,C 180,E1 -22040.249,E2 -22040.249} C_VEL
LIN {X 0,Y 190.708,Z 586.378,A -85,B 0,C 180,E1 -22041.977,E2 -22041.977} C_VEL
LIN {X 0,Y 188.172,Z 587.48,A -85,B 0,C 180,E1 -22044.861,E2 -22044.861} C_VEL
LIN {X 0,Y 186.256,Z 587.736,A -85,B 0,C 180,E1 -22047.238,E2 -22047.238} C_VEL
LIN {X 0,Y 185.752,Z 587.719,A -85,B 0,C 180,E1 -22049.069,E2 -22049.069} C_VEL
LIN {X 0,Y 185.875,Z 587.685,A -85,B 0,C 180,E1 -22049.681,E2 -22049.681} C_VEL
LIN {X 0,Y 185.989,Z 587.688,A -85,B 0,C 180,E1 -22050,E2 -22050} C_VEL
LIN {X 0,Y 184.954,Z 586.024,A -85,B 0,C 180,E1 -22054.358,E2 -22054.358} C_VEL
LIN {X 0,Y 184.48,Z 583.448,A -85,B 0,C 180,E1 -22057.902,E2 -22057.902} C_VEL
LIN {X 0,Y 184.517,Z 578.938,A -85,B 0,C 180,E1 -22062.092,E2 -22062.092} C_VEL
LIN {X 0,Y 185.224,Z 574.101,A -85,B 0,C 180,E1 -22065.402,E2 -22065.402} C_VEL
LIN {X 0,Y 186.602,Z 568.025,A -85,B 0,C 180,E1 -22068.671,E2 -22068.671} C_VEL
LIN {X 0,Y 188.863,Z 560.537,A -85,B 0,C 180,E1 -22071.846,E2 -22071.846} C_VEL
LIN {X 0,Y 190.233,Z 554.53,A -85,B 0,C 180,E1 -22073.978,E2 -22073.978} C_VEL
LIN {X 0,Y 191.864,Z 544.45,A -85,B 0,C 180,E1 -22076.955,E2 -22076.955} C_VEL
LIN {X 0,Y 193.16,Z 533.429,A -85,B 0,C 180,E1 -22079.624,E2 -22079.624} C_VEL
LIN {X 0,Y 193.824,Z 523.056,A -85,B 0,C 180,E1 -22081.719,E2 -22081.719} C_VEL
LIN {X 0,Y 193.901,Z 511.376,A -85,B 0,C 180,E1 -22083.716,E2 -22083.716} C_VEL
LIN {X 0,Y 193.319,Z 500.15,A -85,B 0,C 180,E1 -22085.358,E2 -22085.358} C_VEL
LIN {X 0,Y 191.635,Z 487.237,A -85,B 0,C 180,E1 -22087.017,E2 -22087.017} C_VEL
LIN {X 0,Y 189.319,Z 474.565,A -85,B 0,C 180,E1 -22088.466,E2 -22088.466} C_VEL
LIN {X 0,Y 189.966,Z 471.859,A -85,B 0,C 180,E1 -22090.348,E2 -22090.348} C_VEL
LIN {X 0,Y 189.35,Z 467.55,A -85,B 0,C 180,E1 -22093.635,E2 -22093.635} C_VEL
LIN {X 0,Y 188.234,Z 461.705,A -85,B 0,C 180,E1 -22098.307,E2 -22098.307} C_VEL
LIN {X 0,Y 187.195,Z 456.155,A -85,B 0,C 180,E1 -22103.08,E2 -22103.08} C_VEL
LIN {X 0,Y 186.323,Z 451.991,A -85,B 0,C 180,E1 -22107.028,E2 -22107.028} C_VEL
LIN {X 0,Y 185.602,Z 448.366,A -85,B 0,C 180,E1 -22110.779,E2 -22110.779} C_VEL
LIN {X 0,Y 185.606,Z 448.366,A -85,B 0,C 180,E1 -22115.385,E2 -22115.385} C_VEL
LIN {X 0,Y 185.711,Z 448.356,A -85,B 0,C 180,E1 -22121.101,E2 -22121.101} C_VEL
LIN {X 0,Y 185.7,Z 448.356,A -85,B 0,C 180,E1 -22124.638,E2 -22124.638} C_VEL
LIN {X 0,Y 185.888,Z 448.332,A -85,B 0,C 180,E1 -22129.418,E2 -22129.418} C_VEL
LIN {X 0,Y 185.947,Z 448.323,A -85,B 0,C 180,E1 -22133.49,E2 -22133.49} C_VEL
LIN {X 0,Y 186.209,Z 448.289,A -85,B 0,C 180,E1 -22137.837,E2 -22137.837} C_VEL
LIN {X 0,Y 186.411,Z 448.266,A -85,B 0,C 180,E1 -22140,E2 -22140} C_VEL
LIN {X 0,Y 185.928,Z 448.32,A -85,B 0,C 180,E1 -22144.336,E2 -22144.336} C_VEL
LIN {X 0,Y 186.03,Z 448.311,A -85,B 0,C 180,E1 -22148.692,E2 -22148.692} C_VEL
LIN {X 0,Y 185.743,Z 448.334,A -85,B 0,C 180,E1 -22153.122,E2 -22153.122} C_VEL
LIN {X 0,Y 185.691,Z 448.349,A -85,B 0,C 180,E1 -22157.625,E2 -22157.625} C_VEL
LIN {X 0,Y 185.597,Z 448.323,A -85,B 0,C 180,E1 -22162.252,E2 -22162.252} C_VEL
LIN {X 0,Y 185.564,Z 448.368,A -85,B 0,C 180,E1 -22167.032,E2 -22167.032} C_VEL
LIN {X 0,Y 185.58,Z 448.364,A -85,B 0,C 180,E1 -22169.493,E2 -22169.493} C_VEL
LIN {X 0,Y 185.52,Z 448.35,A -85,B 0,C 180,E1 -22174.628,E2 -22174.628} C_VEL
LIN {X 0,Y 185.545,Z 448.371,A -85,B 0,C 180,E1 -22177.305,E2 -22177.305} C_VEL
LIN {X 0,Y 185.486,Z 448.373,A -85,B 0,C 180,E1 -22180.731,E2 -22180.731} C_VEL
LIN {X 0,Y 185.482,Z 448.377,A -85,B 0,C 180,E1 -22186.048,E2 -22186.048} C_VEL
LIN {X 0,Y 185.491,Z 448.375,A -85,B 0,C 180,E1 -22189.902,E2 -22189.902} C_VEL
LIN {X 0,Y 185.557,Z 448.361,A -85,B 0,C 180,E1 -22194.719,E2 -22194.719} C_VEL
LIN {X 0,Y 185.582,Z 448.542,A -85,B 0,C 180,E1 -22195.232,E2 -22195.232} C_VEL
LIN {X 0,Y 185.882,Z 449.803,A -85,B 0,C 180,E1 -22195.45,E2 -22195.45} C_VEL
LIN {X 0,Y 189.245,Z 455.976,A -85,B 0,C 180,E1 -22197.039,E2 -22197.039} C_VEL
LIN {X 0,Y 193.979,Z 466.713,A -85,B 0,C 180,E1 -22199.795,E2 -22199.795} C_VEL
LIN {X 0,Y 197.024,Z 475.318,A -85,B 0,C 180,E1 -22202.084,E2 -22202.084} C_VEL
LIN {X 0,Y 199.492,Z 484.569,A -85,B 0,C 180,E1 -22204.698,E2 -22204.698} C_VEL
LIN {X 0,Y 200.29,Z 488.341,A -85,B 0,C 180,E1 -22205.829,E2 -22205.829} C_VEL
LIN {X 0,Y 200.297,Z 489.685,A -85,B 0,C 180,E1 -22206.202,E2 -22206.202} C_VEL
LIN {X 0,Y 197.58,Z 499.083,A -85,B 0,C 180,E1 -22208.618,E2 -22208.618} C_VEL
LIN {X 0,Y 195.18,Z 506.765,A -85,B 0,C 180,E1 -22211.091,E2 -22211.091} C_VEL
LIN {X 0,Y 192.704,Z 514.255,A -85,B 0,C 180,E1 -22214.126,E2 -22214.126} C_VEL
LIN {X 0,Y 190.739,Z 520.25,A -85,B 0,C 180,E1 -22217.228,E2 -22217.228} C_VEL
LIN {X 0,Y 189.033,Z 525.032,A -85,B 0,C 180,E1 -22220.369,E2 -22220.369} C_VEL
LIN {X 0,Y 187.631,Z 528.738,A -85,B 0,C 180,E1 -22223.549,E2 -22223.549} C_VEL
LIN {X 0,Y 186.575,Z 532.145,A -85,B 0,C 180,E1 -22227.842,E2 -22227.842} C_VEL
LIN {X 0,Y 186.39,Z 533.867,A -85,B 0,C 180,E1 -22232.161,E2 -22232.161} C_VEL
LIN {X 0,Y 186.466,Z 534.158,A -85,B 0,C 180,E1 -22236.493,E2 -22236.493} C_VEL
LIN {X 0,Y 187.02,Z 533.666,A -85,B 0,C 180,E1 -22238.646,E2 -22238.646} C_VEL
LIN {X 0,Y 188.863,Z 531.491,A -85,B 0,C 180,E1 -22242.902,E2 -22242.902} C_VEL
LIN {X 0,Y 190.741,Z 528.245,A -85,B 0,C 180,E1 -22246.664,E2 -22246.664} C_VEL
LIN {X 0,Y 193.051,Z 523.715,A -85,B 0,C 180,E1 -22250.234,E2 -22250.234} C_VEL
LIN {X 0,Y 195.441,Z 518.545,A -85,B 0,C 180,E1 -22253.301,E2 -22253.301} C_VEL
LIN {X 0,Y 198.249,Z 512.034,A -85,B 0,C 180,E1 -22256.304,E2 -22256.304} C_VEL
LIN {X 0,Y 201.601,Z 503.895,A -85,B 0,C 180,E1 -22259.213,E2 -22259.213} C_VEL
LIN {X 0,Y 203.984,Z 497.287,A -85,B 0,C 180,E1 -22261.119,E2 -22261.119} C_VEL
LIN {X 0,Y 203.89,Z 494.29,A -85,B 0,C 180,E1 -22262.124,E2 -22262.124} C_VEL
LIN {X 0,Y 202.029,Z 485.667,A -85,B 0,C 180,E1 -22265.074,E2 -22265.074} C_VEL
LIN {X 0,Y 199.267,Z 476.651,A -85,B 0,C 180,E1 -22267.985,E2 -22267.985} C_VEL
LIN {X 0,Y 195.483,Z 467.107,A -85,B 0,C 180,E1 -22270.974,E2 -22270.974} C_VEL
LIN {X 0,Y 190.588,Z 457.595,A -85,B 0,C 180,E1 -22274.021,E2 -22274.021} C_VEL
LIN {X 0,Y 187.33,Z 452.317,A -85,B 0,C 180,E1 -22275.801,E2 -22275.801} C_VEL
LIN {X 0,Y 185.823,Z 449.834,A -85,B 0,C 180,E1 -22276.618,E2 -22276.618} C_VEL
LIN {X 0,Y 185.463,Z 448.377,A -85,B 0,C 180,E1 -22276.991,E2 -22276.991} C_VEL
LIN {X 0,Y 185.493,Z 448.374,A -85,B 0,C 180,E1 -22279.901,E2 -22279.901} C_VEL
LIN {X 0,Y 185.547,Z 448.371,A -85,B 0,C 180,E1 -22282.696,E2 -22282.696} C_VEL
LIN {X 0,Y 185.549,Z 448.366,A -85,B 0,C 180,E1 -22287.975,E2 -22287.975} C_VEL
LIN {X 0,Y 185.586,Z 448.365,A -85,B 0,C 180,E1 -22290.576,E2 -22290.576} C_VEL
LIN {X 0,Y 185.583,Z 448.363,A -85,B 0,C 180,E1 -22295.381,E2 -22295.381} C_VEL
LIN {X 0,Y 185.773,Z 448.339,A -85,B 0,C 180,E1 -22299.516,E2 -22299.516} C_VEL
LIN {X 0,Y 188.566,Z 461.372,A -85,B 0,C 180,E1 -22301.53,E2 -22301.53} C_VEL
LIN {X 0,Y 189.336,Z 465.046,A -85,B 0,C 180,E1 -22302.167,E2 -22302.167} C_VEL
LIN {X 0,Y 188.209,Z 477.339,A -85,B 0,C 180,E1 -22304.57,E2 -22304.57} C_VEL
LIN {X 0,Y 187.109,Z 489.161,A -85,B 0,C 180,E1 -22307.4,E2 -22307.4} C_VEL
LIN {X 0,Y 186.122,Z 500.686,A -85,B 0,C 180,E1 -22310.765,E2 -22310.765} C_VEL
LIN {X 0,Y 185.269,Z 511.101,A -85,B 0,C 180,E1 -22314.558,E2 -22314.558} C_VEL
LIN {X 0,Y 185.272,Z 518.525,A -85,B 0,C 180,E1 -22317.826,E2 -22317.826} C_VEL
LIN {X 0,Y 185.713,Z 524.748,A -85,B 0,C 180,E1 -22321.084,E2 -22321.084} C_VEL
LIN {X 0,Y 186.768,Z 531.386,A -85,B 0,C 180,E1 -22325.398,E2 -22325.398} C_VEL
LIN {X 0,Y 188.723,Z 536.442,A -85,B 0,C 180,E1 -22329.647,E2 -22329.647} C_VEL
LIN {X 0,Y 190.992,Z 539.251,A -85,B 0,C 180,E1 -22332.755,E2 -22332.755} C_VEL
LIN {X 0,Y 194.899,Z 541.724,A -85,B 0,C 180,E1 -22336.767,E2 -22336.767} C_VEL
LIN {X 0,Y 199.679,Z 542.86,A -85,B 0,C 180,E1 -22340.607,E2 -22340.607} C_VEL
LIN {X 0,Y 205.34,Z 542.647,A -85,B 0,C 180,E1 -22344.25,E2 -22344.25} C_VEL
LIN {X 0,Y 211.888,Z 541.094,A -85,B 0,C 180,E1 -22347.668,E2 -22347.668} C_VEL
LIN {X 0,Y 219.239,Z 538.228,A -85,B 0,C 180,E1 -22350.857,E2 -22350.857} C_VEL
LIN {X 0,Y 227.334,Z 533.912,A -85,B 0,C 180,E1 -22353.812,E2 -22353.812} C_VEL
LIN {X 0,Y 231.62,Z 531.221,A -85,B 0,C 180,E1 -22355.206,E2 -22355.206} C_VEL
LIN {X 0,Y 233.44,Z 530.073,A -85,B 0,C 180,E1 -22357.022,E2 -22357.022} C_VEL
LIN {X 0,Y 233.407,Z 530.59,A -85,B 0,C 180,E1 -22359.221,E2 -22359.221} C_VEL
LIN {X 0,Y 232.441,Z 532.406,A -85,B 0,C 180,E1 -22361.696,E2 -22361.696} C_VEL
LIN {X 0,Y 230.566,Z 534.662,A -85,B 0,C 180,E1 -22362.982,E2 -22362.982} C_VEL
LIN {X 0,Y 224.193,Z 541.929,A -85,B 0,C 180,E1 -22366.396,E2 -22366.396} C_VEL
LIN {X 0,Y 217.81,Z 549.36,A -85,B 0,C 180,E1 -22369.809,E2 -22369.809} C_VEL
LIN {X 0,Y 211.423,Z 556.423,A -85,B 0,C 180,E1 -22373.248,E2 -22373.248} C_VEL
LIN {X 0,Y 203.061,Z 564.252,A -85,B 0,C 180,E1 -22377.556,E2 -22377.556} C_VEL
LIN {X 0,Y 197.274,Z 569.326,A -85,B 0,C 180,E1 -22381.252,E2 -22381.252} C_VEL
LIN {X 0,Y 193.283,Z 572.392,A -85,B 0,C 180,E1 -22384.129,E2 -22384.129} C_VEL
LIN {X 0,Y 188.625,Z 575.798,A -85,B 0,C 180,E1 -22388.666,E2 -22388.666} C_VEL
LIN {X 0,Y 185.9,Z 577.806,A -85,B 0,C 180,E1 -22393.528,E2 -22393.528} C_VEL
LIN {X 0,Y 185.691,Z 578.237,A -85,B 0,C 180,E1 -22394.073,E2 -22394.073} C_VEL
LIN {X 0,Y 184.485,Z 582.533,A -85,B 0,C 180,E1 -22397.905,E2 -22397.905} C_VEL
LIN {X 0,Y 184.382,Z 585.835,A -85,B 0,C 180,E1 -22402.318,E2 -22402.318} C_VEL
LIN {X 0,Y 184.908,Z 587.248,A -85,B 0,C 180,E1 -22405.64,E2 -22405.64} C_VEL
LIN {X 0,Y 185.875,Z 587.685,A -85,B 0,C 180,E1 -22409.681,E2 -22409.681} C_VEL
LIN {X 0,Y 185.801,Z 587.535,A -85,B 0,C 180,E1 -22410.873,E2 -22410.873} C_VEL
LIN {X 0,Y 184.976,Z 587.12,A -85,B 0,C 180,E1 -22412.043,E2 -22412.043} C_VEL
LIN {X 0,Y 182.088,Z 585.723,A -85,B 0,C 180,E1 -22414.309,E2 -22414.309} C_VEL
LIN {X 0,Y 178.899,Z 583.802,A -85,B 0,C 180,E1 -22416.635,E2 -22416.635} C_VEL
LIN {X 0,Y 177.463,Z 582.172,A -85,B 0,C 180,E1 -22418.469,E2 -22418.469} C_VEL
LIN {X 0,Y 177.331,Z 581.603,A -85,B 0,C 180,E1 -22419.1,E2 -22419.1} C_VEL
LIN {X 0,Y 177.497,Z 577.835,A -85,B 0,C 180,E1 -22422.578,E2 -22422.578} C_VEL
LIN {X 0,Y 178.305,Z 572.977,A -85,B 0,C 180,E1 -22426.016,E2 -22426.016} C_VEL
LIN {X 0,Y 179.85,Z 566.885,A -85,B 0,C 180,E1 -22429.399,E2 -22429.399} C_VEL
LIN {X 0,Y 182.234,Z 559.37,A -85,B 0,C 180,E1 -22432.684,E2 -22432.684} C_VEL
LIN {X 0,Y 183.535,Z 553.303,A -85,B 0,C 180,E1 -22434.911,E2 -22434.911} C_VEL
LIN {X 0,Y 185.257,Z 543.173,A -85,B 0,C 180,E1 -22437.999,E2 -22437.999} C_VEL
LIN {X 0,Y 186.591,Z 532.897,A -85,B 0,C 180,E1 -22440.575,E2 -22440.575} C_VEL
LIN {X 0,Y 187.405,Z 521.763,A -85,B 0,C 180,E1 -22442.916,E2 -22442.916} C_VEL
LIN {X 0,Y 187.495,Z 510.096,A -85,B 0,C 180,E1 -22444.99,E2 -22444.99} C_VEL
LIN {X 0,Y 186.759,Z 497.532,A -85,B 0,C 180,E1 -22446.904,E2 -22446.904} C_VEL
LIN {X 0,Y 184.945,Z 484.145,A -85,B 0,C 180,E1 -22448.686,E2 -22448.686} C_VEL
LIN {X 0,Y 182.785,Z 473.398,A -85,B 0,C 180,E1 -22450.013,E2 -22450.013} C_VEL
LIN {X 0,Y 182.743,Z 470.935,A -85,B 0,C 180,E1 -22451.906,E2 -22451.906} C_VEL
LIN {X 0,Y 181.829,Z 466.051,A -85,B 0,C 180,E1 -22455.915,E2 -22455.915} C_VEL
LIN {X 0,Y 180.643,Z 459.571,A -85,B 0,C 180,E1 -22461.502,E2 -22461.502} C_VEL
LIN {X 0,Y 179.898,Z 455.709,A -85,B 0,C 180,E1 -22465.124,E2 -22465.124} C_VEL
LIN {X 0,Y 178.899,Z 451.127,A -85,B 0,C 180,E1 -22469.798,E2 -22469.798} C_VEL
LIN {X 0,Y 178.58,Z 449.238,A -85,B 0,C 180,E1 -22471.979,E2 -22471.979} C_VEL
LIN {X 0,Y 178.53,Z 449.248,A -85,B 0,C 180,E1 -22476.818,E2 -22476.818} C_VEL
LIN {X 0,Y 178.68,Z 449.233,A -85,B 0,C 180,E1 -22481.66,E2 -22481.66} C_VEL
LIN {X 0,Y 178.66,Z 449.234,A -85,B 0,C 180,E1 -22486.348,E2 -22486.348} C_VEL
LIN {X 0,Y 178.91,Z 449.201,A -85,B 0,C 180,E1 -22490.96,E2 -22490.96} C_VEL
LIN {X 0,Y 179.154,Z 449.168,A -85,B 0,C 180,E1 -22497.752,E2 -22497.752} C_VEL
LIN {X 0,Y 179.373,Z 449.142,A -85,B 0,C 180,E1 -22500,E2 -22500} C_VEL
LIN {X 0,Y 178.877,Z 449.198,A -85,B 0,C 180,E1 -22504.507,E2 -22504.507} C_VEL
LIN {X 0,Y 178.979,Z 449.189,A -85,B 0,C 180,E1 -22509.037,E2 -22509.037} C_VEL
LIN {X 0,Y 178.667,Z 449.216,A -85,B 0,C 180,E1 -22513.652,E2 -22513.652} C_VEL
LIN {X 0,Y 178.624,Z 449.215,A -85,B 0,C 180,E1 -22519.217,E2 -22519.217} C_VEL
LIN {X 0,Y 178.535,Z 449.226,A -85,B 0,C 180,E1 -22525.125,E2 -22525.125} C_VEL
LIN {X 0,Y 178.524,Z 449.238,A -85,B 0,C 180,E1 -22529.994,E2 -22529.994} C_VEL
LIN {X 0,Y 178.497,Z 449.22,A -85,B 0,C 180,E1 -22534.225,E2 -22534.225} C_VEL
LIN {X 0,Y 178.419,Z 449.258,A -85,B 0,C 180,E1 -22539.069,E2 -22539.069} C_VEL
LIN {X 0,Y 178.413,Z 449.26,A -85,B 0,C 180,E1 -22542.042,E2 -22542.042} C_VEL
LIN {X 0,Y 178.404,Z 449.253,A -85,B 0,C 180,E1 -22545.161,E2 -22545.161} C_VEL
LIN {X 0,Y 178.417,Z 449.249,A -85,B 0,C 180,E1 -22548.455,E2 -22548.455} C_VEL
LIN {X 0,Y 178.542,Z 449.417,A -85,B 0,C 180,E1 -22553.501,E2 -22553.501} C_VEL
LIN {X 0,Y 179.334,Z 451.741,A -85,B 0,C 180,E1 -22553.996,E2 -22553.996} C_VEL
LIN {X 0,Y 183.868,Z 460.136,A -85,B 0,C 180,E1 -22556.372,E2 -22556.372} C_VEL
LIN {X 0,Y 188.209,Z 470.3,A -85,B 0,C 180,E1 -22559.189,E2 -22559.189} C_VEL
LIN {X 0,Y 190.824,Z 477.983,A -85,B 0,C 180,E1 -22561.394,E2 -22561.394} C_VEL
LIN {X 0,Y 193.084,Z 487.012,A -85,B 0,C 180,E1 -22564.102,E2 -22564.102} C_VEL
LIN {X 0,Y 193.809,Z 491.283,A -85,B 0,C 180,E1 -22565.448,E2 -22565.448} C_VEL
LIN {X 0,Y 191.073,Z 500.291,A -85,B 0,C 180,E1 -22567.852,E2 -22567.852} C_VEL
LIN {X 0,Y 188.162,Z 509.258,A -85,B 0,C 180,E1 -22570.925,E2 -22570.925} C_VEL
LIN {X 0,Y 185.566,Z 516.482,A -85,B 0,C 180,E1 -22574.063,E2 -22574.063} C_VEL
LIN {X 0,Y 183.297,Z 523.092,A -85,B 0,C 180,E1 -22577.826,E2 -22577.826} C_VEL
LIN {X 0,Y 181.621,Z 527.479,A -85,B 0,C 180,E1 -22581.096,E2 -22581.096} C_VEL
LIN {X 0,Y 180.654,Z 529.809,A -85,B 0,C 180,E1 -22583.298,E2 -22583.298} C_VEL
LIN {X 0,Y 179.979,Z 531.708,A -85,B 0,C 180,E1 -22585.521,E2 -22585.521} C_VEL
LIN {X 0,Y 179.556,Z 533.193,A -85,B 0,C 180,E1 -22587.757,E2 -22587.757} C_VEL
LIN {X 0,Y 179.366,Z 534.893,A -85,B 0,C 180,E1 -22592.246,E2 -22592.246} C_VEL
LIN {X 0,Y 179.479,Z 535.164,A -85,B 0,C 180,E1 -22596.747,E2 -22596.747} C_VEL
LIN {X 0,Y 180.957,Z 533.748,A -85,B 0,C 180,E1 -22601.198,E2 -22601.198} C_VEL
LIN {X 0,Y 182.017,Z 532.462,A -85,B 0,C 180,E1 -22603.396,E2 -22603.396} C_VEL
LIN {X 0,Y 184.012,Z 529.199,A -85,B 0,C 180,E1 -22607.285,E2 -22607.285} C_VEL
LIN {X 0,Y 186.468,Z 524.637,A -85,B 0,C 180,E1 -22610.981,E2 -22610.981} C_VEL
LIN {X 0,Y 189.444,Z 518.469,A -85,B 0,C 180,E1 -22614.668,E2 -22614.668} C_VEL
LIN {X 0,Y 192.477,Z 511.701,A -85,B 0,C 180,E1 -22617.746,E2 -22617.746} C_VEL
LIN {X 0,Y 195.894,Z 503.631,A -85,B 0,C 180,E1 -22620.566,E2 -22620.566} C_VEL
LIN {X 0,Y 197.329,Z 499.855,A -85,B 0,C 180,E1 -22621.691,E2 -22621.691} C_VEL
LIN {X 0,Y 197.719,Z 498.137,A -85,B 0,C 180,E1 -22622.221,E2 -22622.221} C_VEL
LIN {X 0,Y 196.454,Z 490.851,A -85,B 0,C 180,E1 -22624.918,E2 -22624.918} C_VEL
LIN {X 0,Y 193.886,Z 481.325,A -85,B 0,C 180,E1 -22628.255,E2 -22628.255} C_VEL
LIN {X 0,Y 190.494,Z 472.044,A -85,B 0,C 180,E1 -22631.385,E2 -22631.385} C_VEL
LIN {X 0,Y 185.981,Z 462.646,A -85,B 0,C 180,E1 -22634.62,E2 -22634.62} C_VEL
LIN {X 0,Y 183.242,Z 457.883,A -85,B 0,C 180,E1 -22636.34,E2 -22636.34} C_VEL
LIN {X 0,Y 179.994,Z 452.909,A -85,B 0,C 180,E1 -22638.245,E2 -22638.245} C_VEL
LIN {X 0,Y 178.644,Z 450.305,A -85,B 0,C 180,E1 -22639.118,E2 -22639.118} C_VEL
LIN {X 0,Y 178.453,Z 449.255,A -85,B 0,C 180,E1 -22639.37,E2 -22639.37} C_VEL
LIN {X 0,Y 178.453,Z 449.25,A -85,B 0,C 180,E1 -22643.79,E2 -22643.79} C_VEL
LIN {X 0,Y 178.495,Z 449.249,A -85,B 0,C 180,E1 -22646.548,E2 -22646.548} C_VEL
LIN {X 0,Y 178.527,Z 449.247,A -85,B 0,C 180,E1 -22650.006,E2 -22650.006} C_VEL
LIN {X 0,Y 178.523,Z 449.244,A -85,B 0,C 180,E1 -22654.886,E2 -22654.886} C_VEL
LIN {X 0,Y 178.734,Z 449.215,A -85,B 0,C 180,E1 -22659.519,E2 -22659.519} C_VEL
LIN {X 0,Y 181.368,Z 461.509,A -85,B 0,C 180,E1 -22661.464,E2 -22661.464} C_VEL
LIN {X 0,Y 182.186,Z 466.255,A -85,B 0,C 180,E1 -22662.314,E2 -22662.314} C_VEL
LIN {X 0,Y 180.97,Z 478.495,A -85,B 0,C 180,E1 -22664.803,E2 -22664.803} C_VEL
LIN {X 0,Y 179.979,Z 489.34,A -85,B 0,C 180,E1 -22667.484,E2 -22667.484} C_VEL
LIN {X 0,Y 178.977,Z 500.826,A -85,B 0,C 180,E1 -22670.963,E2 -22670.963} C_VEL
LIN {X 0,Y 178.238,Z 510.036,A -85,B 0,C 180,E1 -22674.342,E2 -22674.342} C_VEL
LIN {X 0,Y 178.197,Z 519.015,A -85,B 0,C 180,E1 -22678.305,E2 -22678.305} C_VEL
LIN {X 0,Y 178.773,Z 526.258,A -85,B 0,C 180,E1 -22682.253,E2 -22682.253} C_VEL
LIN {X 0,Y 180.05,Z 532.885,A -85,B 0,C 180,E1 -22686.725,E2 -22686.725} C_VEL
LIN {X 0,Y 182.443,Z 537.896,A -85,B 0,C 180,E1 -22691.105,E2 -22691.105} C_VEL
LIN {X 0,Y 186.072,Z 541.46,A -85,B 0,C 180,E1 -22695.331,E2 -22695.331} C_VEL
LIN {X 0,Y 190.51,Z 543.679,A -85,B 0,C 180,E1 -22699.391,E2 -22699.391} C_VEL
LIN {X 0,Y 195.99,Z 544.503,A -85,B 0,C 180,E1 -22703.231,E2 -22703.231} C_VEL
LIN {X 0,Y 202.373,Z 544.043,A -85,B 0,C 180,E1 -22706.837,E2 -22706.837} C_VEL
LIN {X 0,Y 209.647,Z 542.269,A -85,B 0,C 180,E1 -22710.188,E2 -22710.188} C_VEL
LIN {X 0,Y 217.711,Z 539.135,A -85,B 0,C 180,E1 -22713.283,E2 -22713.283} C_VEL
LIN {X 0,Y 226.425,Z 534.687,A -85,B 0,C 180,E1 -22716.194,E2 -22716.194} C_VEL
LIN {X 0,Y 227.665,Z 534.302,A -85,B 0,C 180,E1 -22718.126,E2 -22718.126} C_VEL
LIN {X 0,Y 227.452,Z 534.875,A -85,B 0,C 180,E1 -22719.423,E2 -22719.423} C_VEL
LIN {X 0,Y 227.082,Z 535.646,A -85,B 0,C 180,E1 -22720.536,E2 -22720.536} C_VEL
LIN {X 0,Y 225.93,Z 537.033,A -85,B 0,C 180,E1 -22721.705,E2 -22721.705} C_VEL
LIN {X 0,Y 219.22,Z 543.789,A -85,B 0,C 180,E1 -22725.145,E2 -22725.145} C_VEL
LIN {X 0,Y 212.484,Z 550.653,A -85,B 0,C 180,E1 -22728.584,E2 -22728.584} C_VEL
LIN {X 0,Y 205.783,Z 557.168,A -85,B 0,C 180,E1 -22732.066,E2 -22732.066} C_VEL
LIN {X 0,Y 197.095,Z 564.383,A -85,B 0,C 180,E1 -22736.447,E2 -22736.447} C_VEL
LIN {X 0,Y 191.06,Z 569.017,A -85,B 0,C 180,E1 -22740.225,E2 -22740.225} C_VEL
LIN {X 0,Y 184.519,Z 573.262,A -85,B 0,C 180,E1 -22745.23,E2 -22745.23} C_VEL
LIN {X 0,Y 180.819,Z 575.453,A -85,B 0,C 180,E1 -22749.524,E2 -22749.524} C_VEL
LIN {X 0,Y 179.094,Z 576.526,A -85,B 0,C 180,E1 -22752.883,E2 -22752.883} C_VEL
LIN {X 0,Y 177.762,Z 580.448,A -85,B 0,C 180,E1 -22756.277,E2 -22756.277} C_VEL
LIN {X 0,Y 177.331,Z 582.527,A -85,B 0,C 180,E1 -22758.57,E2 -22758.57} C_VEL
LIN {X 0,Y 177.327,Z 584.96,A -85,B 0,C 180,E1 -22762.231,E2 -22762.231} C_VEL
LIN {X 0,Y 177.806,Z 586.234,A -85,B 0,C 180,E1 -22765.465,E2 -22765.465} C_VEL
LIN {X 0,Y 178.899,Z 586.661,A -85,B 0,C 180,E1 -22769.926,E2 -22769.926} C_VEL
LIN {X 0,Y 178.268,Z 586.013,A -85,B 0,C 180,E1 -22772.259,E2 -22772.259} C_VEL
LIN {X 0,Y 177.854,Z 584.971,A -85,B 0,C 180,E1 -22774.532,E2 -22774.532} C_VEL
LIN {X 0,Y 177.408,Z 582.595,A -85,B 0,C 180,E1 -22777.957,E2 -22777.957} C_VEL
LIN {X 0,Y 177.331,Z 581.603,A -85,B 0,C 180,E1 -22779.1,E2 -22779.1} C_VEL
LIN {X 0,Y 176.676,Z 579.811,A -85,B 0,C 180,E1 -22780.91,E2 -22780.91} C_VEL
LIN {X 0,Y 174.155,Z 576.162,A -85,B 0,C 180,E1 -22783.811,E2 -22783.811} C_VEL
LIN {X 0,Y 172.054,Z 571.84,A -85,B 0,C 180,E1 -22786.696,E2 -22786.696} C_VEL
LIN {X 0,Y 172.081,Z 568.99,A -85,B 0,C 180,E1 -22788.427,E2 -22788.427} C_VEL
LIN {X 0,Y 174.554,Z 561.548,A -85,B 0,C 180,E1 -22792.175,E2 -22792.175} C_VEL
LIN {X 0,Y 176.313,Z 555.258,A -85,B 0,C 180,E1 -22794.742,E2 -22794.742} C_VEL
LIN {X 0,Y 177.935,Z 546.804,A -85,B 0,C 180,E1 -22797.651,E2 -22797.651} C_VEL
LIN {X 0,Y 179.546,Z 536.46,A -85,B 0,C 180,E1 -22800.588,E2 -22800.588} C_VEL
LIN {X 0,Y 180.628,Z 526.245,A -85,B 0,C 180,E1 -22803.005,E2 -22803.005} C_VEL
LIN {X 0,Y 181.167,Z 515.578,A -85,B 0,C 180,E1 -22805.154,E2 -22805.154} C_VEL
LIN {X 0,Y 180.987,Z 503.91,A -85,B 0,C 180,E1 -22807.181,E2 -22807.181} C_VEL
LIN {X 0,Y 179.792,Z 490.8,A -85,B 0,C 180,E1 -22809.17,E2 -22809.17} C_VEL
LIN {X 0,Y 177.802,Z 479.159,A -85,B 0,C 180,E1 -22810.767,E2 -22810.767} C_VEL
LIN {X 0,Y 176.915,Z 475.897,A -85,B 0,C 180,E1 -22811.246,E2 -22811.246} C_VEL
LIN {X 0,Y 175.753,Z 472.204,A -85,B 0,C 180,E1 -22811.823,E2 -22811.823} C_VEL
LIN {X 0,Y 174.637,Z 466.345,A -85,B 0,C 180,E1 -22816.832,E2 -22816.832} C_VEL
LIN {X 0,Y 173.742,Z 461.334,A -85,B 0,C 180,E1 -22821.366,E2 -22821.366} C_VEL
LIN {X 0,Y 172.983,Z 457.254,A -85,B 0,C 180,E1 -22825.334,E2 -22825.334} C_VEL
LIN {X 0,Y 171.911,Z 452.265,A -85,B 0,C 180,E1 -22830.622,E2 -22830.622} C_VEL
LIN {X 0,Y 171.483,Z 450.121,A -85,B 0,C 180,E1 -22833.204,E2 -22833.204} C_VEL
LIN {X 0,Y 171.484,Z 450.127,A -85,B 0,C 180,E1 -22838.356,E2 -22838.356} C_VEL
LIN {X 0,Y 171.61,Z 450.112,A -85,B 0,C 180,E1 -22840.876,E2 -22840.876} C_VEL
LIN {X 0,Y 171.581,Z 450.116,A -85,B 0,C 180,E1 -22845.773,E2 -22845.773} C_VEL
LIN {X 0,Y 171.847,Z 450.082,A -85,B 0,C 180,E1 -22850.585,E2 -22850.585} C_VEL
LIN {X 0,Y 171.817,Z 450.081,A -85,B 0,C 180,E1 -22855.308,E2 -22855.308} C_VEL
LIN {X 0,Y 172.336,Z 450.019,A -85,B 0,C 180,E1 -22860,E2 -22860} C_VEL
LIN {X 0,Y 171.827,Z 450.075,A -85,B 0,C 180,E1 -22864.693,E2 -22864.693} C_VEL
LIN {X 0,Y 171.905,Z 450.07,A -85,B 0,C 180,E1 -22869.412,E2 -22869.412} C_VEL
LIN {X 0,Y 171.583,Z 450.102,A -85,B 0,C 180,E1 -22874.227,E2 -22874.227} C_VEL
LIN {X 0,Y 171.545,Z 450.092,A -85,B 0,C 180,E1 -22879.563,E2 -22879.563} C_VEL
LIN {X 0,Y 171.47,Z 450.112,A -85,B 0,C 180,E1 -22885.617,E2 -22885.617} C_VEL
LIN {X 0,Y 171.442,Z 450.113,A -85,B 0,C 180,E1 -22890.587,E2 -22890.587} C_VEL
LIN {X 0,Y 171.407,Z 450.109,A -85,B 0,C 180,E1 -22895.032,E2 -22895.032} C_VEL
LIN {X 0,Y 171.381,Z 450.136,A -85,B 0,C 180,E1 -22898.817,E2 -22898.817} C_VEL
LIN {X 0,Y 171.329,Z 450.133,A -85,B 0,C 180,E1 -22904.215,E2 -22904.215} C_VEL
LIN {X 0,Y 171.349,Z 450.131,A -85,B 0,C 180,E1 -22908.986,E2 -22908.986} C_VEL
LIN {X 0,Y 171.395,Z 450.125,A -85,B 0,C 180,E1 -22911.522,E2 -22911.522} C_VEL
LIN {X 0,Y 172.434,Z 452.96,A -85,B 0,C 180,E1 -22912.202,E2 -22912.202} C_VEL
LIN {X 0,Y 176.186,Z 459.466,A -85,B 0,C 180,E1 -22914.249,E2 -22914.249} C_VEL
LIN {X 0,Y 180.311,Z 468.424,A -85,B 0,C 180,E1 -22916.929,E2 -22916.929} C_VEL
LIN {X 0,Y 183.218,Z 476.252,A -85,B 0,C 180,E1 -22919.286,E2 -22919.286} C_VEL
LIN {X 0,Y 185.846,Z 485.363,A -85,B 0,C 180,E1 -22922.138,E2 -22922.138} C_VEL
LIN {X 0,Y 187.349,Z 492.914,A -85,B 0,C 180,E1 -22924.65,E2 -22924.65} C_VEL
LIN {X 0,Y 184.602,Z 501.495,A -85,B 0,C 180,E1 -22927.032,E2 -22927.032} C_VEL
LIN {X 0,Y 181.555,Z 510.419,A -85,B 0,C 180,E1 -22930.202,E2 -22930.202} C_VEL
LIN {X 0,Y 178.861,Z 517.612,A -85,B 0,C 180,E1 -22933.449,E2 -22933.449} C_VEL
LIN {X 0,Y 176.447,Z 524.192,A -85,B 0,C 180,E1 -22937.346,E2 -22937.346} C_VEL
LIN {X 0,Y 174.707,Z 528.556,A -85,B 0,C 180,E1 -22940.741,E2 -22940.741} C_VEL
LIN {X 0,Y 173.681,Z 530.88,A -85,B 0,C 180,E1 -22943.028,E2 -22943.028} C_VEL
LIN {X 0,Y 172.978,Z 532.77,A -85,B 0,C 180,E1 -22945.34,E2 -22945.34} C_VEL
LIN {X 0,Y 172.537,Z 534.24,A -85,B 0,C 180,E1 -22947.666,E2 -22947.666} C_VEL
LIN {X 0,Y 172.343,Z 535.918,A -85,B 0,C 180,E1 -22952.338,E2 -22952.338} C_VEL
LIN {X 0,Y 172.496,Z 536.168,A -85,B 0,C 180,E1 -22957.021,E2 -22957.021} C_VEL
LIN {X 0,Y 174.066,Z 534.729,A -85,B 0,C 180,E1 -22961.647,E2 -22961.647} C_VEL
LIN {X 0,Y 175.185,Z 533.434,A -85,B 0,C 180,E1 -22963.929,E2 -22963.929} C_VEL
LIN {X 0,Y 177.31,Z 530.148,A -85,B 0,C 180,E1 -22967.956,E2 -22967.956} C_VEL
LIN {X 0,Y 179.919,Z 525.559,A -85,B 0,C 180,E1 -22971.783,E2 -22971.783} C_VEL
LIN {X 0,Y 183.051,Z 519.372,A -85,B 0,C 180,E1 -22975.591,E2 -22975.591} C_VEL
LIN {X 0,Y 186.276,Z 512.567,A -85,B 0,C 180,E1 -22978.754,E2 -22978.754} C_VEL
LIN {X 0,Y 189.877,Z 504.46,A -85,B 0,C 180,E1 -22981.644,E2 -22981.644} C_VEL
LIN {X 0,Y 191.255,Z 500.848,A -85,B 0,C 180,E1 -22982.759,E2 -22982.759} C_VEL
LIN {X 0,Y 190.525,Z 494.919,A -85,B 0,C 180,E1 -22985.1,E2 -22985.1} C_VEL
LIN {X 0,Y 188.451,Z 486.044,A -85,B 0,C 180,E1 -22988.448,E2 -22988.448} C_VEL
LIN {X 0,Y 185.829,Z 478.08,A -85,B 0,C 180,E1 -22991.367,E2 -22991.367} C_VEL
LIN {X 0,Y 183.011,Z 471.247,A -85,B 0,C 180,E1 -22993.861,E2 -22993.861} C_VEL
LIN {X 0,Y 178.374,Z 462.387,A -85,B 0,C 180,E1 -22997.283,E2 -22997.283} C_VEL
LIN {X 0,Y 174.523,Z 455.623,A -85,B 0,C 180,E1 -22999.951,E2 -22999.951} C_VEL
LIN {X 0,Y 173.53,Z 454.377,A -85,B 0,C 180,E1 -23000.543,E2 -23000.543} C_VEL
LIN {X 0,Y 171.91,Z 451.992,A -85,B 0,C 180,E1 -23001.596,E2 -23001.596} C_VEL
LIN {X 0,Y 171.435,Z 450.129,A -85,B 0,C 180,E1 -23002.146,E2 -23002.146} C_VEL
LIN {X 0,Y 171.431,Z 450.124,A -85,B 0,C 180,E1 -23007.795,E2 -23007.795} C_VEL
LIN {X 0,Y 171.452,Z 450.126,A -85,B 0,C 180,E1 -23010.534,E2 -23010.534} C_VEL
LIN {X 0,Y 171.465,Z 450.12,A -85,B 0,C 180,E1 -23015.802,E2 -23015.802} C_VEL
LIN {X 0,Y 171.717,Z 450.199,A -85,B 0,C 180,E1 -23019.549,E2 -23019.549} C_VEL
LIN {X 0,Y 174.273,Z 462.09,A -85,B 0,C 180,E1 -23021.483,E2 -23021.483} C_VEL
LIN {X 0,Y 175.047,Z 465.86,A -85,B 0,C 180,E1 -23022.173,E2 -23022.173} C_VEL
LIN {X 0,Y 174.038,Z 476.971,A -85,B 0,C 180,E1 -23024.482,E2 -23024.482} C_VEL
LIN {X 0,Y 172.842,Z 489.552,A -85,B 0,C 180,E1 -23027.659,E2 -23027.659} C_VEL
LIN {X 0,Y 171.874,Z 500.896,A -85,B 0,C 180,E1 -23031.179,E2 -23031.179} C_VEL
LIN {X 0,Y 171.152,Z 510.316,A -85,B 0,C 180,E1 -23034.698,E2 -23034.698} C_VEL
LIN {X 0,Y 171.205,Z 519.344,A -85,B 0,C 180,E1 -23038.824,E2 -23038.824} C_VEL
LIN {X 0,Y 171.699,Z 525.82,A -85,B 0,C 180,E1 -23042.346,E2 -23042.346} C_VEL
LIN {X 0,Y 173.012,Z 532.812,A -85,B 0,C 180,E1 -23046.999,E2 -23046.999} C_VEL
LIN {X 0,Y 175.49,Z 538.213,A -85,B 0,C 180,E1 -23051.551,E2 -23051.551} C_VEL
LIN {X 0,Y 179.294,Z 542.167,A -85,B 0,C 180,E1 -23055.925,E2 -23055.925} C_VEL
LIN {X 0,Y 183.917,Z 544.739,A -85,B 0,C 180,E1 -23060.115,E2 -23060.115} C_VEL
LIN {X 0,Y 189.647,Z 545.983,A -85,B 0,C 180,E1 -23064.057,E2 -23064.057} C_VEL
LIN {X 0,Y 196.309,Z 545.948,A -85,B 0,C 180,E1 -23067.736,E2 -23067.736} C_VEL
LIN {X 0,Y 203.858,Z 544.598,A -85,B 0,C 180,E1 -23071.139,E2 -23071.139} C_VEL
LIN {X 0,Y 212.235,Z 541.965,A -85,B 0,C 180,E1 -23074.259,E2 -23074.259} C_VEL
LIN {X 0,Y 216.657,Z 540.17,A -85,B 0,C 180,E1 -23075.724,E2 -23075.724} C_VEL
LIN {X 0,Y 220.89,Z 538.233,A -85,B 0,C 180,E1 -23077.194,E2 -23077.194} C_VEL
LIN {X 0,Y 221.38,Z 538.728,A -85,B 0,C 180,E1 -23079.414,E2 -23079.414} C_VEL
LIN {X 0,Y 220.992,Z 539.373,A -85,B 0,C 180,E1 -23080.248,E2 -23080.248} C_VEL
LIN {X 0,Y 219.627,Z 540.702,A -85,B 0,C 180,E1 -23081.236,E2 -23081.236} C_VEL
LIN {X 0,Y 212.541,Z 547.03,A -85,B 0,C 180,E1 -23084.689,E2 -23084.689} C_VEL
LIN {X 0,Y 203.732,Z 554.841,A -85,B 0,C 180,E1 -23089.047,E2 -23089.047} C_VEL
LIN {X 0,Y 198.403,Z 559.236,A -85,B 0,C 180,E1 -23091.69,E2 -23091.69} C_VEL
LIN {X 0,Y 189.527,Z 565.509,A -85,B 0,C 180,E1 -23096.204,E2 -23096.204} C_VEL
LIN {X 0,Y 183.413,Z 569.462,A -85,B 0,C 180,E1 -23100.123,E2 -23100.123} C_VEL
LIN {X 0,Y 178.099,Z 572.348,A -85,B 0,C 180,E1 -23104.273,E2 -23104.273} C_VEL
LIN {X 0,Y 174.211,Z 574.178,A -85,B 0,C 180,E1 -23108.71,E2 -23108.71} C_VEL
LIN {X 0,Y 172.6,Z 574.82,A -85,B 0,C 180,E1 -23111.604,E2 -23111.604} C_VEL
LIN {X 0,Y 170.841,Z 579.473,A -85,B 0,C 180,E1 -23115.71,E2 -23115.71} C_VEL
LIN {X 0,Y 170.336,Z 581.543,A -85,B 0,C 180,E1 -23118.094,E2 -23118.094} C_VEL
LIN {X 0,Y 170.262,Z 584.093,A -85,B 0,C 180,E1 -23122.164,E2 -23122.164} C_VEL
LIN {X 0,Y 170.707,Z 585.22,A -85,B 0,C 180,E1 -23125.276,E2 -23125.276} C_VEL
LIN {X 0,Y 171.174,Z 585.632,A -85,B 0,C 180,E1 -23127.646,E2 -23127.646} C_VEL
LIN {X 0,Y 171.862,Z 585.634,A -85,B 0,C 180,E1 -23129.999,E2 -23129.999} C_VEL
LIN {X 0,Y 170.758,Z 583.917,A -85,B 0,C 180,E1 -23134.721,E2 -23134.721} C_VEL
LIN {X 0,Y 170.29,Z 580.918,A -85,B 0,C 180,E1 -23139.005,E2 -23139.005} C_VEL
LIN {X 0,Y 170.506,Z 576.732,A -85,B 0,C 180,E1 -23143.103,E2 -23143.103} C_VEL
LIN {X 0,Y 171.413,Z 571.852,A -85,B 0,C 180,E1 -23146.678,E2 -23146.678} C_VEL
LIN {X 0,Y 172.081,Z 568.99,A -85,B 0,C 180,E1 -23148.427,E2 -23148.427} C_VEL
LIN {X 0,Y 172.292,Z 565.977,A -85,B 0,C 180,E1 -23150.126,E2 -23150.126} C_VEL
LIN {X 0,Y 171.15,Z 560.584,A -85,B 0,C 180,E1 -23152.89,E2 -23152.89} C_VEL
LIN {X 0,Y 170.073,Z 554.599,A -85,B 0,C 180,E1 -23155.558,E2 -23155.558} C_VEL
LIN {X 0,Y 170.383,Z 550.649,A -85,B 0,C 180,E1 -23157.063,E2 -23157.063} C_VEL
LIN {X 0,Y 172.38,Z 540.249,A -85,B 0,C 180,E1 -23160.426,E2 -23160.426} C_VEL
LIN {X 0,Y 173.786,Z 530.28,A -85,B 0,C 180,E1 -23163.089,E2 -23163.089} C_VEL
LIN {X 0,Y 174.685,Z 519.352,A -85,B 0,C 180,E1 -23165.558,E2 -23165.558} C_VEL
LIN {X 0,Y 174.878,Z 507.318,A -85,B 0,C 180,E1 -23167.874,E2 -23167.874} C_VEL
LIN {X 0,Y 174.165,Z 495.047,A -85,B 0,C 180,E1 -23169.942,E2 -23169.942} C_VEL
LIN {X 0,Y 172.461,Z 482.464,A -85,B 0,C 180,E1 -23171.846,E2 -23171.846} C_VEL
LIN {X 0,Y 171.456,Z 478.827,A -85,B 0,C 180,E1 -23172.454,E2 -23172.454} C_VEL
LIN {X 0,Y 170.285,Z 475.765,A -85,B 0,C 180,E1 -23173.037,E2 -23173.037} C_VEL
LIN {X 0,Y 168.58,Z 472.052,A -85,B 0,C 180,E1 -23173.801,E2 -23173.801} C_VEL
LIN {X 0,Y 168.31,Z 470.82,A -85,B 0,C 180,E1 -23174.029,E2 -23174.029} C_VEL
LIN {X 0,Y 167.239,Z 465.24,A -85,B 0,C 180,E1 -23179.15,E2 -23179.15} C_VEL
LIN {X 0,Y 166.411,Z 460.511,A -85,B 0,C 180,E1 -23183.754,E2 -23183.754} C_VEL
LIN {X 0,Y 165.31,Z 455.297,A -85,B 0,C 180,E1 -23189.325,E2 -23189.325} C_VEL
LIN {X 0,Y 164.909,Z 452.954,A -85,B 0,C 180,E1 -23192.044,E2 -23192.044} C_VEL
LIN {X 0,Y 164.418,Z 451.005,A -85,B 0,C 180,E1 -23194.695,E2 -23194.695} C_VEL
LIN {X 0,Y 164.52,Z 450.996,A -85,B 0,C 180,E1 -23200.017,E2 -23200.017} C_VEL
LIN {X 0,Y 164.531,Z 450.993,A -85,B 0,C 180,E1 -23205.15,E2 -23205.15} C_VEL
LIN {X 0,Y 164.767,Z 450.963,A -85,B 0,C 180,E1 -23210.177,E2 -23210.177} C_VEL
LIN {X 0,Y 164.831,Z 450.953,A -85,B 0,C 180,E1 -23212.651,E2 -23212.651} C_VEL
LIN {X 0,Y 165.049,Z 450.925,A -85,B 0,C 180,E1 -23217.56,E2 -23217.56} C_VEL
LIN {X 0,Y 165.298,Z 450.895,A -85,B 0,C 180,E1 -23220,E2 -23220} C_VEL
LIN {X 0,Y 164.841,Z 450.94,A -85,B 0,C 180,E1 -23227.115,E2 -23227.115} C_VEL
LIN {X 0,Y 164.751,Z 450.958,A -85,B 0,C 180,E1 -23231.146,E2 -23231.146} C_VEL
LIN {X 0,Y 164.485,Z 450.991,A -85,B 0,C 180,E1 -23237.403,E2 -23237.403} C_VEL
LIN {X 0,Y 164.474,Z 450.965,A -85,B 0,C 180,E1 -23239.99,E2 -23239.99} C_VEL
LIN {X 0,Y 164.394,Z 450.997,A -85,B 0,C 180,E1 -23246.135,E2 -23246.135} C_VEL
LIN {X 0,Y 164.377,Z 450.984,A -85,B 0,C 180,E1 -23251.229,E2 -23251.229} C_VEL
LIN {X 0,Y 164.337,Z 451.01,A -85,B 0,C 180,E1 -23256.779,E2 -23256.779} C_VEL
LIN {X 0,Y 164.301,Z 451.011,A -85,B 0,C 180,E1 -23259.914,E2 -23259.914} C_VEL
LIN {X 0,Y 164.28,Z 451.015,A -85,B 0,C 180,E1 -23263.343,E2 -23263.343} C_VEL
LIN {X 0,Y 164.318,Z 451.006,A -85,B 0,C 180,E1 -23268.925,E2 -23268.925} C_VEL
LIN {X 0,Y 164.298,Z 451.01,A -85,B 0,C 180,E1 -23269.31,E2 -23269.31} C_VEL
LIN {X 0,Y 165.153,Z 453.622,A -85,B 0,C 180,E1 -23269.995,E2 -23269.995} C_VEL
LIN {X 0,Y 166.684,Z 455.473,A -85,B 0,C 180,E1 -23270.769,E2 -23270.769} C_VEL
LIN {X 0,Y 171.646,Z 465.263,A -85,B 0,C 180,E1 -23273.967,E2 -23273.967} C_VEL
LIN {X 0,Y 175.267,Z 473.677,A -85,B 0,C 180,E1 -23276.707,E2 -23276.707} C_VEL
LIN {X 0,Y 178.247,Z 482.674,A -85,B 0,C 180,E1 -23279.665,E2 -23279.665} C_VEL
LIN {X 0,Y 180.298,Z 491.728,A -85,B 0,C 180,E1 -23282.764,E2 -23282.764} C_VEL
LIN {X 0,Y 180.831,Z 494.569,A -85,B 0,C 180,E1 -23283.788,E2 -23283.788} C_VEL
LIN {X 0,Y 178.171,Z 502.694,A -85,B 0,C 180,E1 -23286.152,E2 -23286.152} C_VEL
LIN {X 0,Y 174.978,Z 511.579,A -85,B 0,C 180,E1 -23289.425,E2 -23289.425} C_VEL
LIN {X 0,Y 172.168,Z 518.744,A -85,B 0,C 180,E1 -23292.786,E2 -23292.786} C_VEL
LIN {X 0,Y 169.61,Z 525.293,A -85,B 0,C 180,E1 -23296.827,E2 -23296.827} C_VEL
LIN {X 0,Y 167.799,Z 529.634,A -85,B 0,C 180,E1 -23300.356,E2 -23300.356} C_VEL
LIN {X 0,Y 166.712,Z 531.951,A -85,B 0,C 180,E1 -23302.735,E2 -23302.735} C_VEL
LIN {X 0,Y 165.979,Z 533.831,A -85,B 0,C 180,E1 -23305.143,E2 -23305.143} C_VEL
LIN {X 0,Y 165.518,Z 535.286,A -85,B 0,C 180,E1 -23307.567,E2 -23307.567} C_VEL
LIN {X 0,Y 165.32,Z 536.944,A -85,B 0,C 180,E1 -23312.437,E2 -23312.437} C_VEL
LIN {X 0,Y 165.341,Z 537.245,A -85,B 0,C 180,E1 -23314.877,E2 -23314.877} C_VEL
LIN {X 0,Y 165.516,Z 537.17,A -85,B 0,C 180,E1 -23317.319,E2 -23317.319} C_VEL
LIN {X 0,Y 167.187,Z 535.71,A -85,B 0,C 180,E1 -23322.134,E2 -23322.134} C_VEL
LIN {X 0,Y 168.369,Z 534.406,A -85,B 0,C 180,E1 -23324.505,E2 -23324.505} C_VEL
LIN {X 0,Y 170.636,Z 531.094,A -85,B 0,C 180,E1 -23328.681,E2 -23328.681} C_VEL
LIN {X 0,Y 173.408,Z 526.481,A -85,B 0,C 180,E1 -23332.646,E2 -23332.646} C_VEL
LIN {X 0,Y 176.713,Z 520.275,A -85,B 0,C 180,E1 -23336.579,E2 -23336.579} C_VEL
LIN {X 0,Y 180.138,Z 513.43,A -85,B 0,C 180,E1 -23339.831,E2 -23339.831} C_VEL
LIN {X 0,Y 183.888,Z 505.363,A -85,B 0,C 180,E1 -23342.773,E2 -23342.773} C_VEL
LIN {X 0,Y 184.77,Z 503.217,A -85,B 0,C 180,E1 -23343.471,E2 -23343.471} C_VEL
LIN {X 0,Y 184.656,Z 499.947,A -85,B 0,C 180,E1 -23344.814,E2 -23344.814} C_VEL
LIN {X 0,Y 183.318,Z 492.644,A -85,B 0,C 180,E1 -23347.837,E2 -23347.837} C_VEL
LIN {X 0,Y 181.294,Z 484.907,A -85,B 0,C 180,E1 -23350.894,E2 -23350.894} C_VEL
LIN {X 0,Y 178.498,Z 477.022,A -85,B 0,C 180,E1 -23353.991,E2 -23353.991} C_VEL
LIN {X 0,Y 174.417,Z 468.379,A -85,B 0,C 180,E1 -23357.551,E2 -23357.551} C_VEL
LIN {X 0,Y 170.423,Z 461.009,A -85,B 0,C 180,E1 -23360.709,E2 -23360.709} C_VEL
LIN {X 0,Y 168.406,Z 458.192,A -85,B 0,C 180,E1 -23362.131,E2 -23362.131} C_VEL
LIN {X 0,Y 167.42,Z 455.98,A -85,B 0,C 180,E1 -23362.969,E2 -23362.969} C_VEL
LIN {X 0,Y 165.297,Z 453.755,A -85,B 0,C 180,E1 -23364.372,E2 -23364.372} C_VEL
LIN {X 0,Y 164.359,Z 451.008,A -85,B 0,C 180,E1 -23365.287,E2 -23365.287} C_VEL
LIN {X 0,Y 164.409,Z 451.003,A -85,B 0,C 180,E1 -23369.138,E2 -23369.138} C_VEL
LIN {X 0,Y 164.413,Z 451.001,A -85,B 0,C 180,E1 -23374.693,E2 -23374.693} C_VEL
LIN {X 0,Y 164.696,Z 451.155,A -85,B 0,C 180,E1 -23379.64,E2 -23379.64} C_VEL
LIN {X 0,Y 167.215,Z 462.917,A -85,B 0,C 180,E1 -23381.625,E2 -23381.625} C_VEL
LIN {X 0,Y 167.931,Z 466.647,A -85,B 0,C 180,E1 -23382.337,E2 -23382.337} C_VEL
LIN {X 0,Y 166.67,Z 479.008,A -85,B 0,C 180,E1 -23385.032,E2 -23385.032} C_VEL
LIN {X 0,Y 165.6,Z 490.448,A -85,B 0,C 180,E1 -23388.059,E2 -23388.059} C_VEL
LIN {X 0,Y 164.745,Z 500.876,A -85,B 0,C 180,E1 -23391.413,E2 -23391.413} C_VEL
LIN {X 0,Y 164.056,Z 511.837,A -85,B 0,C 180,E1 -23395.7,E2 -23395.7} C_VEL
LIN {X 0,Y 164.3,Z 520.831,A -85,B 0,C 180,E1 -23400,E2 -23400} C_VEL
LIN {X 0,Y 164.905,Z 527.206,A -85,B 0,C 180,E1 -23403.665,E2 -23403.665} C_VEL
LIN {X 0,Y 165.981,Z 532.607,A -85,B 0,C 180,E1 -23407.297,E2 -23407.297} C_VEL
LIN {X 0,Y 168.543,Z 538.404,A -85,B 0,C 180,E1 -23412.034,E2 -23412.034} C_VEL
LIN {X 0,Y 172.513,Z 542.711,A -85,B 0,C 180,E1 -23416.569,E2 -23416.569} C_VEL
LIN {X 0,Y 177.353,Z 545.696,A -85,B 0,C 180,E1 -23420.894,E2 -23420.894} C_VEL
LIN {X 0,Y 183.332,Z 547.366,A -85,B 0,C 180,E1 -23424.941,E2 -23424.941} C_VEL
LIN {X 0,Y 190.258,Z 547.718,A -85,B 0,C 180,E1 -23428.699,E2 -23428.699} C_VEL
LIN {X 0,Y 198.099,Z 546.826,A -85,B 0,C 180,E1 -23432.151,E2 -23432.151} C_VEL
LIN {X 0,Y 206.783,Z 544.682,A -85,B 0,C 180,E1 -23435.295,E2 -23435.295} C_VEL
LIN {X 0,Y 211.363,Z 543.12,A -85,B 0,C 180,E1 -23436.763,E2 -23436.763} C_VEL
LIN {X 0,Y 214.961,Z 541.898,A -85,B 0,C 180,E1 -23438.31,E2 -23438.31} C_VEL
LIN {X 0,Y 214.768,Z 542.662,A -85,B 0,C 180,E1 -23439.781,E2 -23439.781} C_VEL
LIN {X 0,Y 213.205,Z 543.977,A -85,B 0,C 180,E1 -23440.697,E2 -23440.697} C_VEL
LIN {X 0,Y 203.918,Z 551.292,A -85,B 0,C 180,E1 -23445.046,E2 -23445.046} C_VEL
LIN {X 0,Y 194.732,Z 558.257,A -85,B 0,C 180,E1 -23449.485,E2 -23449.485} C_VEL
LIN {X 0,Y 185.393,Z 564.238,A -85,B 0,C 180,E1 -23454.013,E2 -23454.013} C_VEL
LIN {X 0,Y 177.273,Z 568.823,A -85,B 0,C 180,E1 -23458.976,E2 -23458.976} C_VEL
LIN {X 0,Y 171.748,Z 571.323,A -85,B 0,C 180,E1 -23463.248,E2 -23463.248} C_VEL
LIN {X 0,Y 167.66,Z 572.807,A -85,B 0,C 180,E1 -23467.835,E2 -23467.835} C_VEL
LIN {X 0,Y 166.147,Z 573.306,A -85,B 0,C 180,E1 -23470.381,E2 -23470.381} C_VEL
LIN {X 0,Y 164.348,Z 577.338,A -85,B 0,C 180,E1 -23473.861,E2 -23473.861} C_VEL
LIN {X 0,Y 163.329,Z 580.555,A -85,B 0,C 180,E1 -23477.575,E2 -23477.575} C_VEL
LIN {X 0,Y 163.198,Z 583.195,A -85,B 0,C 180,E1 -23482.086,E2 -23482.086} C_VEL
LIN {X 0,Y 163.614,Z 584.207,A -85,B 0,C 180,E1 -23485.071,E2 -23485.071} C_VEL
LIN {X 0,Y 164.089,Z 584.615,A -85,B 0,C 180,E1 -23487.545,E2 -23487.545} C_VEL
LIN {X 0,Y 164.799,Z 584.606,A -85,B 0,C 180,E1 -23489.999,E2 -23489.999} C_VEL
LIN {X 0,Y 163.667,Z 582.864,A -85,B 0,C 180,E1 -23494.926,E2 -23494.926} C_VEL
LIN {X 0,Y 163.281,Z 580.858,A -85,B 0,C 180,E1 -23498.121,E2 -23498.121} C_VEL
LIN {X 0,Y 163.343,Z 576.99,A -85,B 0,C 180,E1 -23502.423,E2 -23502.423} C_VEL
LIN {X 0,Y 164.133,Z 572.474,A -85,B 0,C 180,E1 -23506.16,E2 -23506.16} C_VEL
LIN {X 0,Y 165.659,Z 566.774,A -85,B 0,C 180,E1 -23509.84,E2 -23509.84} C_VEL
LIN {X 0,Y 168.093,Z 560.012,A -85,B 0,C 180,E1 -23513.272,E2 -23513.272} C_VEL
LIN {X 0,Y 169.645,Z 554.042,A -85,B 0,C 180,E1 -23515.784,E2 -23515.784} C_VEL
LIN {X 0,Y 170.383,Z 550.649,A -85,B 0,C 180,E1 -23517.063,E2 -23517.063} C_VEL
LIN {X 0,Y 170.611,Z 546.651,A -85,B 0,C 180,E1 -23518.515,E2 -23518.515} C_VEL
LIN {X 0,Y 169.218,Z 540.022,A -85,B 0,C 180,E1 -23520.962,E2 -23520.962} C_VEL
LIN {X 0,Y 167.626,Z 533.045,A -85,B 0,C 180,E1 -23523.337,E2 -23523.337} C_VEL
LIN {X 0,Y 167.525,Z 528.437,A -85,B 0,C 180,E1 -23524.631,E2 -23524.631} C_VEL
LIN {X 0,Y 168.458,Z 517.565,A -85,B 0,C 180,E1 -23527.159,E2 -23527.159} C_VEL
LIN {X 0,Y 168.688,Z 505.619,A -85,B 0,C 180,E1 -23529.547,E2 -23529.547} C_VEL
LIN {X 0,Y 168.009,Z 493.693,A -85,B 0,C 180,E1 -23531.662,E2 -23531.662} C_VEL
LIN {X 0,Y 166.552,Z 483.18,A -85,B 0,C 180,E1 -23533.399,E2 -23533.399} C_VEL
LIN {X 0,Y 165.11,Z 479.436,A -85,B 0,C 180,E1 -23534.229,E2 -23534.229} C_VEL
LIN {X 0,Y 163.089,Z 474.718,A -85,B 0,C 180,E1 -23535.288,E2 -23535.288} C_VEL
LIN {X 0,Y 161.179,Z 470.955,A -85,B 0,C 180,E1 -23536.219,E2 -23536.219} C_VEL
LIN {X 0,Y 160.783,Z 469.371,A -85,B 0,C 180,E1 -23536.542,E2 -23536.542} C_VEL
LIN {X 0,Y 159.761,Z 463.535,A -85,B 0,C 180,E1 -23542.357,E2 -23542.357} C_VEL
LIN {X 0,Y 158.867,Z 459.037,A -85,B 0,C 180,E1 -23547.195,E2 -23547.195} C_VEL
LIN {X 0,Y 157.897,Z 454.247,A -85,B 0,C 180,E1 -23552.897,E2 -23552.897} C_VEL
LIN {X 0,Y 157.322,Z 451.89,A -85,B 0,C 180,E1 -23556.294,E2 -23556.294} C_VEL
LIN {X 0,Y 157.446,Z 451.878,A -85,B 0,C 180,E1 -23559.616,E2 -23559.616} C_VEL
LIN {X 0,Y 157.464,Z 451.874,A -85,B 0,C 180,E1 -23564.467,E2 -23564.467} C_VEL
LIN {X 0,Y 157.689,Z 451.844,A -85,B 0,C 180,E1 -23569.731,E2 -23569.731} C_VEL
LIN {X 0,Y 157.767,Z 451.833,A -85,B 0,C 180,E1 -23572.32,E2 -23572.32} C_VEL
LIN {X 0,Y 158.26,Z 451.772,A -85,B 0,C 180,E1 -23580,E2 -23580} C_VEL
LIN {X 0,Y 157.822,Z 451.817,A -85,B 0,C 180,E1 -23587.678,E2 -23587.678} C_VEL
LIN {X 0,Y 157.68,Z 451.836,A -85,B 0,C 180,E1 -23591.315,E2 -23591.315} C_VEL
LIN {X 0,Y 157.457,Z 451.868,A -85,B 0,C 180,E1 -23595.534,E2 -23595.534} C_VEL
LIN {X 0,Y 157.37,Z 451.837,A -85,B 0,C 180,E1 -23600.933,E2 -23600.933} C_VEL
LIN {X 0,Y 157.316,Z 451.883,A -85,B 0,C 180,E1 -23606.686,E2 -23606.686} C_VEL
LIN {X 0,Y 157.279,Z 451.856,A -85,B 0,C 180,E1 -23612.427,E2 -23612.427} C_VEL
LIN {X 0,Y 157.296,Z 451.883,A -85,B 0,C 180,E1 -23616.464,E2 -23616.464} C_VEL
LIN {X 0,Y 157.214,Z 451.9,A -85,B 0,C 180,E1 -23622.11,E2 -23622.11} C_VEL
LIN {X 0,Y 157.269,Z 452.02,A -85,B 0,C 180,E1 -23626.908,E2 -23626.908} C_VEL
LIN {X 0,Y 158.27,Z 454.764,A -85,B 0,C 180,E1 -23627.712,E2 -23627.712} C_VEL
LIN {X 0,Y 159.632,Z 456.325,A -85,B 0,C 180,E1 -23628.457,E2 -23628.457} C_VEL
LIN {X 0,Y 160.436,Z 458.247,A -85,B 0,C 180,E1 -23629.081,E2 -23629.081} C_VEL
LIN {X 0,Y 163.793,Z 464.033,A -85,B 0,C 180,E1 -23631.289,E2 -23631.289} C_VEL
LIN {X 0,Y 167.301,Z 471.585,A -85,B 0,C 180,E1 -23633.977,E2 -23633.977} C_VEL
LIN {X 0,Y 170.626,Z 480.387,A -85,B 0,C 180,E1 -23637.083,E2 -23637.083} C_VEL
LIN {X 0,Y 172.985,Z 489.248,A -85,B 0,C 180,E1 -23640.241,E2 -23640.241} C_VEL
LIN {X 0,Y 174.182,Z 495.531,A -85,B 0,C 180,E1 -23642.583,E2 -23642.583} C_VEL
LIN {X 0,Y 174.281,Z 496.992,A -85,B 0,C 180,E1 -23643.135,E2 -23643.135} C_VEL
LIN {X 0,Y 171.182,Z 505.483,A -85,B 0,C 180,E1 -23645.761,E2 -23645.761} C_VEL
LIN {X 0,Y 167.946,Z 514.057,A -85,B 0,C 180,E1 -23649.164,E2 -23649.164} C_VEL
LIN {X 0,Y 165.045,Z 520.929,A -85,B 0,C 180,E1 -23652.658,E2 -23652.658} C_VEL
LIN {X 0,Y 162.787,Z 526.392,A -85,B 0,C 180,E1 -23656.264,E2 -23656.264} C_VEL
LIN {X 0,Y 160.896,Z 530.712,A -85,B 0,C 180,E1 -23659.938,E2 -23659.938} C_VEL
LIN {X 0,Y 159.748,Z 533.022,A -85,B 0,C 180,E1 -23662.416,E2 -23662.416} C_VEL
LIN {X 0,Y 158.981,Z 534.892,A -85,B 0,C 180,E1 -23664.928,E2 -23664.928} C_VEL
LIN {X 0,Y 158.499,Z 536.329,A -85,B 0,C 180,E1 -23667.459,E2 -23667.459} C_VEL
LIN {X 0,Y 158.297,Z 537.969,A -85,B 0,C 180,E1 -23672.545,E2 -23672.545} C_VEL
LIN {X 0,Y 158.336,Z 538.262,A -85,B 0,C 180,E1 -23675.094,E2 -23675.094} C_VEL
LIN {X 0,Y 158.542,Z 538.171,A -85,B 0,C 180,E1 -23677.643,E2 -23677.643} C_VEL
LIN {X 0,Y 160.321,Z 536.691,A -85,B 0,C 180,E1 -23682.662,E2 -23682.662} C_VEL
LIN {X 0,Y 161.572,Z 535.378,A -85,B 0,C 180,E1 -23685.129,E2 -23685.129} C_VEL
LIN {X 0,Y 163.951,Z 532.082,A -85,B 0,C 180,E1 -23689.426,E2 -23689.426} C_VEL
LIN {X 0,Y 166.936,Z 527.405,A -85,B 0,C 180,E1 -23693.576,E2 -23693.576} C_VEL
LIN {X 0,Y 170.439,Z 521.177,A -85,B 0,C 180,E1 -23697.639,E2 -23697.639} C_VEL
LIN {X 0,Y 174.069,Z 514.292,A -85,B 0,C 180,E1 -23700.983,E2 -23700.983} C_VEL
LIN {X 0,Y 177.92,Z 506.358,A -85,B 0,C 180,E1 -23703.95,E2 -23703.95} C_VEL
LIN {X 0,Y 178.432,Z 505.204,A -85,B 0,C 180,E1 -23704.332,E2 -23704.332} C_VEL
LIN {X 0,Y 178.383,Z 502.483,A -85,B 0,C 180,E1 -23705.53,E2 -23705.53} C_VEL
LIN {X 0,Y 177.273,Z 495.585,A -85,B 0,C 180,E1 -23708.603,E2 -23708.603} C_VEL
LIN {X 0,Y 175.741,Z 488.99,A -85,B 0,C 180,E1 -23711.425,E2 -23711.425} C_VEL
LIN {X 0,Y 173.218,Z 481.224,A -85,B 0,C 180,E1 -23714.723,E2 -23714.723} C_VEL
LIN {X 0,Y 169.527,Z 472.861,A -85,B 0,C 180,E1 -23718.447,E2 -23718.447} C_VEL
LIN {X 0,Y 166.14,Z 466.224,A -85,B 0,C 180,E1 -23721.521,E2 -23721.521} C_VEL
LIN {X 0,Y 163.514,Z 461.695,A -85,B 0,C 180,E1 -23723.772,E2 -23723.772} C_VEL
LIN {X 0,Y 161.293,Z 458.633,A -85,B 0,C 180,E1 -23725.56,E2 -23725.56} C_VEL
LIN {X 0,Y 160.682,Z 457.085,A -85,B 0,C 180,E1 -23726.179,E2 -23726.179} C_VEL
LIN {X 0,Y 158.389,Z 454.86,A -85,B 0,C 180,E1 -23727.919,E2 -23727.919} C_VEL
LIN {X 0,Y 157.435,Z 452.345,A -85,B 0,C 180,E1 -23728.92,E2 -23728.92} C_VEL
LIN {X 0,Y 157.376,Z 451.878,A -85,B 0,C 180,E1 -23729.098,E2 -23729.098} C_VEL
LIN {X 0,Y 157.319,Z 451.888,A -85,B 0,C 180,E1 -23733.465,E2 -23733.465} C_VEL
LIN {X 0,Y 157.637,Z 452.012,A -85,B 0,C 180,E1 -23739.725,E2 -23739.725} C_VEL
LIN {X 0,Y 160.16,Z 463.74,A -85,B 0,C 180,E1 -23741.781,E2 -23741.781} C_VEL
LIN {X 0,Y 160.774,Z 467.41,A -85,B 0,C 180,E1 -23742.51,E2 -23742.51} C_VEL
LIN {X 0,Y 159.51,Z 479.801,A -85,B 0,C 180,E1 -23745.325,E2 -23745.325} C_VEL
LIN {X 0,Y 158.394,Z 491.11,A -85,B 0,C 180,E1 -23748.487,E2 -23748.487} C_VEL
LIN {X 0,Y 157.655,Z 500.707,A -85,B 0,C 180,E1 -23751.669,E2 -23751.669} C_VEL
LIN {X 0,Y 157.03,Z 510.4,A -85,B 0,C 180,E1 -23755.507,E2 -23755.507} C_VEL
LIN {X 0,Y 157.226,Z 519.825,A -85,B 0,C 180,E1 -23760,E2 -23760} C_VEL
LIN {X 0,Y 157.834,Z 526.581,A -85,B 0,C 180,E1 -23763.829,E2 -23763.829} C_VEL
LIN {X 0,Y 159.532,Z 533.917,A -85,B 0,C 180,E1 -23768.869,E2 -23768.869} C_VEL
LIN {X 0,Y 162.536,Z 539.746,A -85,B 0,C 180,E1 -23773.757,E2 -23773.757} C_VEL
LIN {X 0,Y 165.731,Z 543.139,A -85,B 0,C 180,E1 -23777.268,E2 -23777.268} C_VEL
LIN {X 0,Y 170.803,Z 546.529,A -85,B 0,C 180,E1 -23781.735,E2 -23781.735} C_VEL
LIN {X 0,Y 177.019,Z 548.583,A -85,B 0,C 180,E1 -23785.895,E2 -23785.895} C_VEL
LIN {X 0,Y 184.234,Z 549.384,A -85,B 0,C 180,E1 -23789.73,E2 -23789.73} C_VEL
LIN {X 0,Y 192.381,Z 548.967,A -85,B 0,C 180,E1 -23793.228,E2 -23793.228} C_VEL
LIN {X 0,Y 201.38,Z 547.261,A -85,B 0,C 180,E1 -23796.39,E2 -23796.39} C_VEL
LIN {X 0,Y 206.107,Z 545.948,A -85,B 0,C 180,E1 -23797.863,E2 -23797.863} C_VEL
LIN {X 0,Y 208.459,Z 545.518,A -85,B 0,C 180,E1 -23799.156,E2 -23799.156} C_VEL
LIN {X 0,Y 204.73,Z 548.133,A -85,B 0,C 180,E1 -23800.955,E2 -23800.955} C_VEL
LIN {X 0,Y 196.99,Z 553.517,A -85,B 0,C 180,E1 -23804.476,E2 -23804.476} C_VEL
LIN {X 0,Y 189.351,Z 558.566,A -85,B 0,C 180,E1 -23808.079,E2 -23808.079} C_VEL
LIN {X 0,Y 181.532,Z 563.012,A -85,B 0,C 180,E1 -23811.724,E2 -23811.724} C_VEL
LIN {X 0,Y 174.446,Z 566.591,A -85,B 0,C 180,E1 -23815.665,E2 -23815.665} C_VEL
LIN {X 0,Y 168.24,Z 569.211,A -85,B 0,C 180,E1 -23819.914,E2 -23819.914} C_VEL
LIN {X 0,Y 162.392,Z 571.025,A -85,B 0,C 180,E1 -23825.345,E2 -23825.345} C_VEL
LIN {X 0,Y 159.903,Z 571.545,A -85,B 0,C 180,E1 -23828.908,E2 -23828.908} C_VEL
LIN {X 0,Y 157.497,Z 576.367,A -85,B 0,C 180,E1 -23833.138,E2 -23833.138} C_VEL
LIN {X 0,Y 156.361,Z 579.571,A -85,B 0,C 180,E1 -23837.012,E2 -23837.012} C_VEL
LIN {X 0,Y 156.144,Z 582.281,A -85,B 0,C 180,E1 -23841.976,E2 -23841.976} C_VEL
LIN {X 0,Y 156.527,Z 583.194,A -85,B 0,C 180,E1 -23844.847,E2 -23844.847} C_VEL
LIN {X 0,Y 157.001,Z 583.597,A -85,B 0,C 180,E1 -23847.434,E2 -23847.434} C_VEL
LIN {X 0,Y 157.736,Z 583.576,A -85,B 0,C 180,E1 -23849.999,E2 -23849.999} C_VEL
LIN {X 0,Y 156.581,Z 581.812,A -85,B 0,C 180,E1 -23855.15,E2 -23855.15} C_VEL
LIN {X 0,Y 156.21,Z 580.003,A -85,B 0,C 180,E1 -23858.194,E2 -23858.194} C_VEL
LIN {X 0,Y 156.359,Z 575.896,A -85,B 0,C 180,E1 -23862.987,E2 -23862.987} C_VEL
LIN {X 0,Y 157.223,Z 571.354,A -85,B 0,C 180,E1 -23866.891,E2 -23866.891} C_VEL
LIN {X 0,Y 158.967,Z 565.646,A -85,B 0,C 180,E1 -23870.712,E2 -23870.712} C_VEL
LIN {X 0,Y 161.512,Z 558.852,A -85,B 0,C 180,E1 -23874.28,E2 -23874.28} C_VEL
LIN {X 0,Y 163.524,Z 550.938,A -85,B 0,C 180,E1 -23877.659,E2 -23877.659} C_VEL
LIN {X 0,Y 165.611,Z 541.038,A -85,B 0,C 180,E1 -23881.094,E2 -23881.094} C_VEL
LIN {X 0,Y 167.329,Z 530.178,A -85,B 0,C 180,E1 -23884.177,E2 -23884.177} C_VEL
LIN {X 0,Y 167.525,Z 528.437,A -85,B 0,C 180,E1 -23884.631,E2 -23884.631} C_VEL
LIN {X 0,Y 167.319,Z 523.82,A -85,B 0,C 180,E1 -23885.887,E2 -23885.887} C_VEL
LIN {X 0,Y 165.245,Z 516.5,A -85,B 0,C 180,E1 -23888.101,E2 -23888.101} C_VEL
LIN {X 0,Y 163.047,Z 508.961,A -85,B 0,C 180,E1 -23890.25,E2 -23890.25} C_VEL
LIN {X 0,Y 162.584,Z 503.942,A -85,B 0,C 180,E1 -23891.359,E2 -23891.359} C_VEL
LIN {X 0,Y 162.005,Z 492.524,A -85,B 0,C 180,E1 -23893.484,E2 -23893.484} C_VEL
LIN {X 0,Y 161.074,Z 486.015,A -85,B 0,C 180,E1 -23894.689,E2 -23894.689} C_VEL
LIN {X 0,Y 158.345,Z 479.055,A -85,B 0,C 180,E1 -23896.422,E2 -23896.422} C_VEL
LIN {X 0,Y 156.452,Z 474.764,A -85,B 0,C 180,E1 -23897.53,E2 -23897.53} C_VEL
LIN {X 0,Y 153.859,Z 469.838,A -85,B 0,C 180,E1 -23898.957,E2 -23898.957} C_VEL
LIN {X 0,Y 153.279,Z 467.894,A -85,B 0,C 180,E1 -23899.42,E2 -23899.42} C_VEL
LIN {X 0,Y 152.44,Z 462.841,A -85,B 0,C 180,E1 -23904.812,E2 -23904.812} C_VEL
LIN {X 0,Y 151.38,Z 457.809,A -85,B 0,C 180,E1 -23910.827,E2 -23910.827} C_VEL
LIN {X 0,Y 150.693,Z 454.554,A -85,B 0,C 180,E1 -23915.182,E2 -23915.182} C_VEL
LIN {X 0,Y 150.313,Z 452.764,A -85,B 0,C 180,E1 -23918.035,E2 -23918.035} C_VEL
LIN {X 0,Y 150.393,Z 452.755,A -85,B 0,C 180,E1 -23920.907,E2 -23920.907} C_VEL
LIN {X 0,Y 150.44,Z 452.749,A -85,B 0,C 180,E1 -23926.492,E2 -23926.492} C_VEL
LIN {X 0,Y 150.611,Z 452.726,A -85,B 0,C 180,E1 -23929.243,E2 -23929.243} C_VEL
LIN {X 0,Y 150.705,Z 452.713,A -85,B 0,C 180,E1 -23931.958,E2 -23931.958} C_VEL
LIN {X 0,Y 151.22,Z 452.649,A -85,B 0,C 180,E1 -23940,E2 -23940} C_VEL
LIN {X 0,Y 150.757,Z 452.699,A -85,B 0,C 180,E1 -23948.04,E2 -23948.04} C_VEL
LIN {X 0,Y 150.615,Z 452.713,A -85,B 0,C 180,E1 -23951.508,E2 -23951.508} C_VEL
LIN {X 0,Y 150.365,Z 452.753,A -85,B 0,C 180,E1 -23956.287,E2 -23956.287} C_VEL
LIN {X 0,Y 150.351,Z 452.71,A -85,B 0,C 180,E1 -23960.793,E2 -23960.793} C_VEL
LIN {X 0,Y 150.246,Z 452.767,A -85,B 0,C 180,E1 -23967.283,E2 -23967.283} C_VEL
LIN {X 0,Y 150.219,Z 452.734,A -85,B 0,C 180,E1 -23972.635,E2 -23972.635} C_VEL
LIN {X 0,Y 150.216,Z 452.773,A -85,B 0,C 180,E1 -23977.462,E2 -23977.462} C_VEL
LIN {X 0,Y 150.141,Z 452.779,A -85,B 0,C 180,E1 -23982.924,E2 -23982.924} C_VEL
LIN {X 0,Y 150.158,Z 452.923,A -85,B 0,C 180,E1 -23984.065,E2 -23984.065} C_VEL
LIN {X 0,Y 151.178,Z 455.689,A -85,B 0,C 180,E1 -23984.981,E2 -23984.981} C_VEL
LIN {X 0,Y 152.587,Z 457.276,A -85,B 0,C 180,E1 -23985.844,E2 -23985.844} C_VEL
LIN {X 0,Y 157.865,Z 466.695,A -85,B 0,C 180,E1 -23989.747,E2 -23989.747} C_VEL
LIN {X 0,Y 161.209,Z 474.035,A -85,B 0,C 180,E1 -23992.611,E2 -23992.611} C_VEL
LIN {X 0,Y 164.429,Z 482.695,A -85,B 0,C 180,E1 -23995.928,E2 -23995.928} C_VEL
LIN {X 0,Y 166.675,Z 491.262,A -85,B 0,C 180,E1 -23999.218,E2 -23999.218} C_VEL
LIN {X 0,Y 167.858,Z 498.508,A -85,B 0,C 180,E1 -24002.114,E2 -24002.114} C_VEL
LIN {X 0,Y 164.238,Z 508.256,A -85,B 0,C 180,E1 -24005.341,E2 -24005.341} C_VEL
LIN {X 0,Y 160.824,Z 516.446,A -85,B 0,C 180,E1 -24008.868,E2 -24008.868} C_VEL
LIN {X 0,Y 158.373,Z 522.049,A -85,B 0,C 180,E1 -24011.903,E2 -24011.903} C_VEL
LIN {X 0,Y 155.981,Z 527.492,A -85,B 0,C 180,E1 -24015.652,E2 -24015.652} C_VEL
LIN {X 0,Y 154.001,Z 531.789,A -85,B 0,C 180,E1 -24019.483,E2 -24019.483} C_VEL
LIN {X 0,Y 152.788,Z 534.092,A -85,B 0,C 180,E1 -24022.069,E2 -24022.069} C_VEL
LIN {X 0,Y 152.008,Z 535.95,A -85,B 0,C 180,E1 -24024.695,E2 -24024.695} C_VEL
LIN {X 0,Y 151.481,Z 537.372,A -85,B 0,C 180,E1 -24027.341,E2 -24027.341} C_VEL
LIN {X 0,Y 151.275,Z 538.995,A -85,B 0,C 180,E1 -24032.663,E2 -24032.663} C_VEL
LIN {X 0,Y 151.334,Z 539.279,A -85,B 0,C 180,E1 -24035.33,E2 -24035.33} C_VEL
LIN {X 0,Y 151.573,Z 539.171,A -85,B 0,C 180,E1 -24037.996,E2 -24037.996} C_VEL
LIN {X 0,Y 153.47,Z 537.672,A -85,B 0,C 180,E1 -24043.237,E2 -24043.237} C_VEL
LIN {X 0,Y 154.796,Z 536.35,A -85,B 0,C 180,E1 -24045.808,E2 -24045.808} C_VEL
LIN {X 0,Y 157.288,Z 533.079,A -85,B 0,C 180,E1 -24050.225,E2 -24050.225} C_VEL
LIN {X 0,Y 160.506,Z 528.329,A -85,B 0,C 180,E1 -24054.581,E2 -24054.581} C_VEL
LIN {X 0,Y 164.233,Z 522.077,A -85,B 0,C 180,E1 -24058.779,E2 -24058.779} C_VEL
LIN {X 0,Y 168.075,Z 515.154,A -85,B 0,C 180,E1 -24062.218,E2 -24062.218} C_VEL
LIN {X 0,Y 172.032,Z 507.355,A -85,B 0,C 180,E1 -24065.207,E2 -24065.207} C_VEL
LIN {X 0,Y 172.26,Z 506.506,A -85,B 0,C 180,E1 -24065.547,E2 -24065.547} C_VEL
LIN {X 0,Y 171.423,Z 499.74,A -85,B 0,C 180,E1 -24068.834,E2 -24068.834} C_VEL
LIN {X 0,Y 170.097,Z 493.007,A -85,B 0,C 180,E1 -24071.95,E2 -24071.95} C_VEL
LIN {X 0,Y 167.978,Z 485.642,A -85,B 0,C 180,E1 -24075.338,E2 -24075.338} C_VEL
LIN {X 0,Y 164.58,Z 477.287,A -85,B 0,C 180,E1 -24079.366,E2 -24079.366} C_VEL
LIN {X 0,Y 160.35,Z 468.888,A -85,B 0,C 180,E1 -24083.722,E2 -24083.722} C_VEL
LIN {X 0,Y 159.066,Z 466.722,A -85,B 0,C 180,E1 -24084.943,E2 -24084.943} C_VEL
LIN {X 0,Y 157.196,Z 463.255,A -85,B 0,C 180,E1 -24086.843,E2 -24086.843} C_VEL
LIN {X 0,Y 155.203,Z 460.91,A -85,B 0,C 180,E1 -24088.617,E2 -24088.617} C_VEL
LIN {X 0,Y 153.867,Z 458.1,A -85,B 0,C 180,E1 -24090.093,E2 -24090.093} C_VEL
LIN {X 0,Y 151.437,Z 455.952,A -85,B 0,C 180,E1 -24092.272,E2 -24092.272} C_VEL
LIN {X 0,Y 150.377,Z 453.307,A -85,B 0,C 180,E1 -24093.611,E2 -24093.611} C_VEL
LIN {X 0,Y 150.281,Z 452.765,A -85,B 0,C 180,E1 -24093.924,E2 -24093.924} C_VEL
LIN {X 0,Y 150.601,Z 452.78,A -85,B 0,C 180,E1 -24099.86,E2 -24099.86} C_VEL
LIN {X 0,Y 153.084,Z 464.281,A -85,B 0,C 180,E1 -24101.947,E2 -24101.947} C_VEL
LIN {X 0,Y 153.591,Z 467.915,A -85,B 0,C 180,E1 -24102.696,E2 -24102.696} C_VEL
LIN {X 0,Y 152.382,Z 480.113,A -85,B 0,C 180,E1 -24105.593,E2 -24105.593} C_VEL
LIN {X 0,Y 151.146,Z 492.727,A -85,B 0,C 180,E1 -24109.281,E2 -24109.281} C_VEL
LIN {X 0,Y 150.398,Z 502.162,A -85,B 0,C 180,E1 -24112.616,E2 -24112.616} C_VEL
LIN {X 0,Y 149.973,Z 513.189,A -85,B 0,C 180,E1 -24117.314,E2 -24117.314} C_VEL
LIN {X 0,Y 150.424,Z 522.311,A -85,B 0,C 180,E1 -24122.008,E2 -24122.008} C_VEL
LIN {X 0,Y 151.491,Z 529.794,A -85,B 0,C 180,E1 -24126.66,E2 -24126.66} C_VEL
LIN {X 0,Y 153.913,Z 536.793,A -85,B 0,C 180,E1 -24131.857,E2 -24131.857} C_VEL
LIN {X 0,Y 157.781,Z 542.26,A -85,B 0,C 180,E1 -24136.829,E2 -24136.829} C_VEL
LIN {X 0,Y 161.497,Z 545.462,A -85,B 0,C 180,E1 -24140.374,E2 -24140.374} C_VEL
LIN {X 0,Y 167.388,Z 548.583,A -85,B 0,C 180,E1 -24144.826,E2 -24144.826} C_VEL
LIN {X 0,Y 174.409,Z 550.455,A -85,B 0,C 180,E1 -24148.917,E2 -24148.917} C_VEL
LIN {X 0,Y 182.386,Z 551.096,A -85,B 0,C 180,E1 -24152.647,E2 -24152.647} C_VEL
LIN {X 0,Y 191.259,Z 550.482,A -85,B 0,C 180,E1 -24156.01,E2 -24156.01} C_VEL
LIN {X 0,Y 200.828,Z 548.695,A -85,B 0,C 180,E1 -24159.043,E2 -24159.043} C_VEL
LIN {X 0,Y 192.01,Z 554.101,A -85,B 0,C 180,E1 -24162.941,E2 -24162.941} C_VEL
LIN {X 0,Y 184.07,Z 558.695,A -85,B 0,C 180,E1 -24166.586,E2 -24166.586} C_VEL
LIN {X 0,Y 175.986,Z 562.692,A -85,B 0,C 180,E1 -24170.285,E2 -24170.285} C_VEL
LIN {X 0,Y 168.615,Z 565.835,A -85,B 0,C 180,E1 -24174.3,E2 -24174.3} C_VEL
LIN {X 0,Y 162.183,Z 568.07,A -85,B 0,C 180,E1 -24178.667,E2 -24178.667} C_VEL
LIN {X 0,Y 156.143,Z 569.459,A -85,B 0,C 180,E1 -24184.184,E2 -24184.184} C_VEL
LIN {X 0,Y 153.792,Z 569.766,A -85,B 0,C 180,E1 -24187.32,E2 -24187.32} C_VEL
LIN {X 0,Y 151.321,Z 574.092,A -85,B 0,C 180,E1 -24191.027,E2 -24191.027} C_VEL
LIN {X 0,Y 149.738,Z 577.608,A -85,B 0,C 180,E1 -24195.039,E2 -24195.039} C_VEL
LIN {X 0,Y 149.052,Z 580.177,A -85,B 0,C 180,E1 -24199.128,E2 -24199.128} C_VEL
LIN {X 0,Y 149.44,Z 582.181,A -85,B 0,C 180,E1 -24204.602,E2 -24204.602} C_VEL
LIN {X 0,Y 149.911,Z 582.578,A -85,B 0,C 180,E1 -24207.312,E2 -24207.312} C_VEL
LIN {X 0,Y 150.643,Z 582.543,A -85,B 0,C 180,E1 -24209.999,E2 -24209.999} C_VEL
LIN {X 0,Y 149.494,Z 580.759,A -85,B 0,C 180,E1 -24215.395,E2 -24215.395} C_VEL
LIN {X 0,Y 149.141,Z 579.142,A -85,B 0,C 180,E1 -24218.276,E2 -24218.276} C_VEL
LIN {X 0,Y 149.181,Z 576.092,A -85,B 0,C 180,E1 -24222.239,E2 -24222.239} C_VEL
LIN {X 0,Y 149.926,Z 571.9,A -85,B 0,C 180,E1 -24226.335,E2 -24226.335} C_VEL
LIN {X 0,Y 151.882,Z 565.554,A -85,B 0,C 180,E1 -24231.015,E2 -24231.015} C_VEL
LIN {X 0,Y 154.608,Z 558.711,A -85,B 0,C 180,E1 -24234.864,E2 -24234.864} C_VEL
LIN {X 0,Y 156.552,Z 551.619,A -85,B 0,C 180,E1 -24238.123,E2 -24238.123} C_VEL
LIN {X 0,Y 158.582,Z 543.042,A -85,B 0,C 180,E1 -24241.381,E2 -24241.381} C_VEL
LIN {X 0,Y 160.561,Z 532.529,A -85,B 0,C 180,E1 -24244.682,E2 -24244.682} C_VEL
LIN {X 0,Y 161.888,Z 522.054,A -85,B 0,C 180,E1 -24247.428,E2 -24247.428} C_VEL
LIN {X 0,Y 162.584,Z 510.069,A -85,B 0,C 180,E1 -24250.116,E2 -24250.116} C_VEL
LIN {X 0,Y 162.584,Z 503.942,A -85,B 0,C 180,E1 -24251.359,E2 -24251.359} C_VEL
LIN {X 0,Y 162.294,Z 500.581,A -85,B 0,C 180,E1 -24252.073,E2 -24252.073} C_VEL
LIN {X 0,Y 160.847,Z 495.993,A -85,B 0,C 180,E1 -24253.306,E2 -24253.306} C_VEL
LIN {X 0,Y 158.667,Z 491.856,A -85,B 0,C 180,E1 -24254.646,E2 -24254.646} C_VEL
LIN {X 0,Y 153.71,Z 483.655,A -85,B 0,C 180,E1 -24257.471,E2 -24257.471} C_VEL
LIN {X 0,Y 152.349,Z 480.623,A -85,B 0,C 180,E1 -24258.361,E2 -24258.361} C_VEL
LIN {X 0,Y 151.162,Z 477.855,A -85,B 0,C 180,E1 -24259.171,E2 -24259.171} C_VEL
LIN {X 0,Y 149.299,Z 473.687,A -85,B 0,C 180,E1 -24260.408,E2 -24260.408} C_VEL
LIN {X 0,Y 148.378,Z 471.994,A -85,B 0,C 180,E1 -24260.983,E2 -24260.983} C_VEL
LIN {X 0,Y 146.376,Z 468.232,A -85,B 0,C 180,E1 -24262.254,E2 -24262.254} C_VEL
LIN {X 0,Y 145.808,Z 466.288,A -85,B 0,C 180,E1 -24262.734,E2 -24262.734} C_VEL
LIN {X 0,Y 145.032,Z 462.055,A -85,B 0,C 180,E1 -24267.789,E2 -24267.789} C_VEL
LIN {X 0,Y 144.273,Z 458.432,A -85,B 0,C 180,E1 -24272.536,E2 -24272.536} C_VEL
LIN {X 0,Y 143.402,Z 453.962,A -85,B 0,C 180,E1 -24279.041,E2 -24279.041} C_VEL
LIN {X 0,Y 143.341,Z 453.634,A -85,B 0,C 180,E1 -24279.928,E2 -24279.928} C_VEL
LIN {X 0,Y 143.365,Z 453.632,A -85,B 0,C 180,E1 -24285.812,E2 -24285.812} C_VEL
LIN {X 0,Y 143.537,Z 453.609,A -85,B 0,C 180,E1 -24288.706,E2 -24288.706} C_VEL
LIN {X 0,Y 143.626,Z 453.596,A -85,B 0,C 180,E1 -24291.559,E2 -24291.559} C_VEL
LIN {X 0,Y 144.179,Z 453.526,A -85,B 0,C 180,E1 -24300,E2 -24300} C_VEL
LIN {X 0,Y 143.676,Z 453.583,A -85,B 0,C 180,E1 -24308.439,E2 -24308.439} C_VEL
LIN {X 0,Y 143.548,Z 453.591,A -85,B 0,C 180,E1 -24311.713,E2 -24311.713} C_VEL
LIN {X 0,Y 143.304,Z 453.63,A -85,B 0,C 180,E1 -24317.114,E2 -24317.114} C_VEL
LIN {X 0,Y 143.277,Z 453.586,A -85,B 0,C 180,E1 -24321.255,E2 -24321.255} C_VEL
LIN {X 0,Y 143.192,Z 453.649,A -85,B 0,C 180,E1 -24327.938,E2 -24327.938} C_VEL
LIN {X 0,Y 143.169,Z 453.61,A -85,B 0,C 180,E1 -24333.436,E2 -24333.436} C_VEL
LIN {X 0,Y 143.077,Z 453.654,A -85,B 0,C 180,E1 -24339.686,E2 -24339.686} C_VEL
LIN {X 0,Y 143.105,Z 453.65,A -85,B 0,C 180,E1 -24340.736,E2 -24340.736} C_VEL
LIN {X 0,Y 144.108,Z 456.504,A -85,B 0,C 180,E1 -24341.788,E2 -24341.788} C_VEL
LIN {X 0,Y 146.336,Z 459.484,A -85,B 0,C 180,E1 -24343.448,E2 -24343.448} C_VEL
LIN {X 0,Y 147.296,Z 461.406,A -85,B 0,C 180,E1 -24344.3,E2 -24344.3} C_VEL
LIN {X 0,Y 148.571,Z 462.987,A -85,B 0,C 180,E1 -24345.2,E2 -24345.2} C_VEL
LIN {X 0,Y 153.208,Z 471.902,A -85,B 0,C 180,E1 -24349.194,E2 -24349.194} C_VEL
LIN {X 0,Y 156.185,Z 479.012,A -85,B 0,C 180,E1 -24352.197,E2 -24352.197} C_VEL
LIN {X 0,Y 159.013,Z 487.55,A -85,B 0,C 180,E1 -24355.735,E2 -24355.735} C_VEL
LIN {X 0,Y 160.77,Z 495.633,A -85,B 0,C 180,E1 -24359.094,E2 -24359.094} C_VEL
LIN {X 0,Y 161.335,Z 499.118,A -85,B 0,C 180,E1 -24360.603,E2 -24360.603} C_VEL
LIN {X 0,Y 161.342,Z 501.018,A -85,B 0,C 180,E1 -24361.37,E2 -24361.37} C_VEL
LIN {X 0,Y 157.898,Z 509.439,A -85,B 0,C 180,E1 -24364.281,E2 -24364.281} C_VEL
LIN {X 0,Y 154.309,Z 517.592,A -85,B 0,C 180,E1 -24367.93,E2 -24367.93} C_VEL
LIN {X 0,Y 151.729,Z 523.169,A -85,B 0,C 180,E1 -24371.081,E2 -24371.081} C_VEL
LIN {X 0,Y 149.194,Z 528.591,A -85,B 0,C 180,E1 -24374.985,E2 -24374.985} C_VEL
LIN {X 0,Y 147.114,Z 532.868,A -85,B 0,C 180,E1 -24378.984,E2 -24378.984} C_VEL
LIN {X 0,Y 145.857,Z 535.159,A -85,B 0,C 180,E1 -24381.689,E2 -24381.689} C_VEL
LIN {X 0,Y 145.035,Z 537.008,A -85,B 0,C 180,E1 -24384.439,E2 -24384.439} C_VEL
LIN {X 0,Y 144.463,Z 538.415,A -85,B 0,C 180,E1 -24387.212,E2 -24387.212} C_VEL
LIN {X 0,Y 144.254,Z 540.02,A -85,B 0,C 180,E1 -24392.793,E2 -24392.793} C_VEL
LIN {X 0,Y 144.335,Z 540.296,A -85,B 0,C 180,E1 -24395.589,E2 -24395.589} C_VEL
LIN {X 0,Y 144.61,Z 540.17,A -85,B 0,C 180,E1 -24398.384,E2 -24398.384} C_VEL
LIN {X 0,Y 146.636,Z 538.653,A -85,B 0,C 180,E1 -24403.866,E2 -24403.866} C_VEL
LIN {X 0,Y 148.043,Z 537.322,A -85,B 0,C 180,E1 -24406.55,E2 -24406.55} C_VEL
LIN {X 0,Y 150.698,Z 534.037,A -85,B 0,C 180,E1 -24411.134,E2 -24411.134} C_VEL
LIN {X 0,Y 154.128,Z 529.253,A -85,B 0,C 180,E1 -24415.671,E2 -24415.671} C_VEL
LIN {X 0,Y 158.099,Z 522.975,A -85,B 0,C 180,E1 -24420.007,E2 -24420.007} C_VEL
LIN {X 0,Y 162.159,Z 516.018,A -85,B 0,C 180,E1 -24423.545,E2 -24423.545} C_VEL
LIN {X 0,Y 165.949,Z 508.796,A -85,B 0,C 180,E1 -24426.422,E2 -24426.422} C_VEL
LIN {X 0,Y 165.261,Z 501.825,A -85,B 0,C 180,E1 -24430.049,E2 -24430.049} C_VEL
LIN {X 0,Y 164.097,Z 495.383,A -85,B 0,C 180,E1 -24433.273,E2 -24433.273} C_VEL
LIN {X 0,Y 161.987,Z 488.048,A -85,B 0,C 180,E1 -24436.97,E2 -24436.97} C_VEL
LIN {X 0,Y 159.292,Z 481.004,A -85,B 0,C 180,E1 -24440.662,E2 -24440.662} C_VEL
LIN {X 0,Y 155.832,Z 473.404,A -85,B 0,C 180,E1 -24444.898,E2 -24444.898} C_VEL
LIN {X 0,Y 152.955,Z 468.398,A -85,B 0,C 180,E1 -24448.102,E2 -24448.102} C_VEL
LIN {X 0,Y 151.055,Z 465.275,A -85,B 0,C 180,E1 -24450.255,E2 -24450.255} C_VEL
LIN {X 0,Y 147.896,Z 460.898,A -85,B 0,C 180,E1 -24453.829,E2 -24453.829} C_VEL
LIN {X 0,Y 147.275,Z 459.214,A -85,B 0,C 180,E1 -24454.796,E2 -24454.796} C_VEL
LIN {X 0,Y 144.866,Z 457.271,A -85,B 0,C 180,E1 -24457.5,E2 -24457.5} C_VEL
LIN {X 0,Y 143.763,Z 454.861,A -85,B 0,C 180,E1 -24459.266,E2 -24459.266} C_VEL
LIN {X 0,Y 143.545,Z 453.597,A -85,B 0,C 180,E1 -24459.854,E2 -24459.854} C_VEL
LIN {X 0,Y 143.596,Z 453.638,A -85,B 0,C 180,E1 -24460.057,E2 -24460.057} C_VEL
LIN {X 0,Y 146.423,Z 466.624,A -85,B 0,C 180,E1 -24462.543,E2 -24462.543} C_VEL
LIN {X 0,Y 145.502,Z 477.118,A -85,B 0,C 180,E1 -24465.027,E2 -24465.027} C_VEL
LIN {X 0,Y 144.397,Z 488.932,A -85,B 0,C 180,E1 -24468.435,E2 -24468.435} C_VEL
LIN {X 0,Y 143.487,Z 499.907,A -85,B 0,C 180,E1 -24472.259,E2 -24472.259} C_VEL
LIN {X 0,Y 142.971,Z 510.01,A -85,B 0,C 180,E1 -24476.477,E2 -24476.477} C_VEL
LIN {X 0,Y 143.334,Z 519.832,A -85,B 0,C 180,E1 -24481.404,E2 -24481.404} C_VEL
LIN {X 0,Y 144.264,Z 527.935,A -85,B 0,C 180,E1 -24486.293,E2 -24486.293} C_VEL
LIN {X 0,Y 146.192,Z 534.661,A -85,B 0,C 180,E1 -24491.086,E2 -24491.086} C_VEL
LIN {X 0,Y 149.799,Z 540.929,A -85,B 0,C 180,E1 -24496.349,E2 -24496.349} C_VEL
LIN {X 0,Y 154.866,Z 545.77,A -85,B 0,C 180,E1 -24501.287,E2 -24501.287} C_VEL
LIN {X 0,Y 161.023,Z 549.318,A -85,B 0,C 180,E1 -24505.878,E2 -24505.878} C_VEL
LIN {X 0,Y 168.323,Z 551.636,A -85,B 0,C 180,E1 -24510.068,E2 -24510.068} C_VEL
LIN {X 0,Y 176.593,Z 552.694,A -85,B 0,C 180,E1 -24513.86,E2 -24513.86} C_VEL
LIN {X 0,Y 185.789,Z 552.542,A -85,B 0,C 180,E1 -24517.246,E2 -24517.246} C_VEL
LIN {X 0,Y 190.697,Z 552.028,A -85,B 0,C 180,E1 -24518.794,E2 -24518.794} C_VEL
LIN {X 0,Y 191.315,Z 552.25,A -85,B 0,C 180,E1 -24519.516,E2 -24519.516} C_VEL
LIN {X 0,Y 182.996,Z 556.603,A -85,B 0,C 180,E1 -24523.138,E2 -24523.138} C_VEL
LIN {X 0,Y 178.933,Z 558.642,A -85,B 0,C 180,E1 -24525.008,E2 -24525.008} C_VEL
LIN {X 0,Y 170.563,Z 562.201,A -85,B 0,C 180,E1 -24528.755,E2 -24528.755} C_VEL
LIN {X 0,Y 162.9,Z 564.927,A -85,B 0,C 180,E1 -24532.842,E2 -24532.842} C_VEL
LIN {X 0,Y 156.206,Z 566.785,A -85,B 0,C 180,E1 -24537.322,E2 -24537.322} C_VEL
LIN {X 0,Y 150.034,Z 567.753,A -85,B 0,C 180,E1 -24542.874,E2 -24542.874} C_VEL
LIN {X 0,Y 147.831,Z 567.991,A -85,B 0,C 180,E1 -24545.605,E2 -24545.605} C_VEL
LIN {X 0,Y 144.604,Z 573.128,A -85,B 0,C 180,E1 -24550.109,E2 -24550.109} C_VEL
LIN {X 0,Y 142.851,Z 576.625,A -85,B 0,C 180,E1 -24554.3,E2 -24554.3} C_VEL
LIN {X 0,Y 142.053,Z 579.177,A -85,B 0,C 180,E1 -24558.585,E2 -24558.585} C_VEL
LIN {X 0,Y 142.355,Z 581.168,A -85,B 0,C 180,E1 -24564.333,E2 -24564.333} C_VEL
LIN {X 0,Y 142.82,Z 581.557,A -85,B 0,C 180,E1 -24567.179,E2 -24567.179} C_VEL
LIN {X 0,Y 143.551,Z 581.509,A -85,B 0,C 180,E1 -24569.999,E2 -24569.999} C_VEL
LIN {X 0,Y 142.39,Z 579.703,A -85,B 0,C 180,E1 -24575.665,E2 -24575.665} C_VEL
LIN {X 0,Y 142.017,Z 577.201,A -85,B 0,C 180,E1 -24579.974,E2 -24579.974} C_VEL
LIN {X 0,Y 142.4,Z 573.702,A -85,B 0,C 180,E1 -24584.286,E2 -24584.286} C_VEL
LIN {X 0,Y 143.535,Z 569.121,A -85,B 0,C 180,E1 -24588.557,E2 -24588.557} C_VEL
LIN {X 0,Y 145.697,Z 563.386,A -85,B 0,C 180,E1 -24592.699,E2 -24592.699} C_VEL
LIN {X 0,Y 148.095,Z 557.546,A -85,B 0,C 180,E1 -24596.038,E2 -24596.038} C_VEL
LIN {X 0,Y 150.536,Z 548.84,A -85,B 0,C 180,E1 -24600.124,E2 -24600.124} C_VEL
LIN {X 0,Y 152.743,Z 539.875,A -85,B 0,C 180,E1 -24603.514,E2 -24603.514} C_VEL
LIN {X 0,Y 154.551,Z 529.959,A -85,B 0,C 180,E1 -24606.644,E2 -24606.644} C_VEL
LIN {X 0,Y 155.818,Z 520.625,A -85,B 0,C 180,E1 -24609.157,E2 -24609.157} C_VEL
LIN {X 0,Y 156.598,Z 508.831,A -85,B 0,C 180,E1 -24611.917,E2 -24611.917} C_VEL
LIN {X 0,Y 156.505,Z 497.358,A -85,B 0,C 180,E1 -24614.301,E2 -24614.301} C_VEL
LIN {X 0,Y 155.961,Z 490.246,A -85,B 0,C 180,E1 -24615.698,E2 -24615.698} C_VEL
LIN {X 0,Y 153.808,Z 483.776,A -85,B 0,C 180,E1 -24617.404,E2 -24617.404} C_VEL
LIN {X 0,Y 152.349,Z 480.623,A -85,B 0,C 180,E1 -24618.361,E2 -24618.361} C_VEL
LIN {X 0,Y 150.748,Z 478.053,A -85,B 0,C 180,E1 -24619.306,E2 -24619.306} C_VEL
LIN {X 0,Y 148.615,Z 476.263,A -85,B 0,C 180,E1 -24620.402,E2 -24620.402} C_VEL
LIN {X 0,Y 142.562,Z 472.318,A -85,B 0,C 180,E1 -24623.602,E2 -24623.602} C_VEL
LIN {X 0,Y 141.375,Z 470.818,A -85,B 0,C 180,E1 -24624.375,E2 -24624.375} C_VEL
LIN {X 0,Y 139.004,Z 466.735,A -85,B 0,C 180,E1 -24626.114,E2 -24626.114} C_VEL
LIN {X 0,Y 138.319,Z 464.563,A -85,B 0,C 180,E1 -24626.784,E2 -24626.784} C_VEL
LIN {X 0,Y 137.429,Z 460.303,A -85,B 0,C 180,E1 -24632.597,E2 -24632.597} C_VEL
LIN {X 0,Y 136.623,Z 456.149,A -85,B 0,C 180,E1 -24638.895,E2 -24638.895} C_VEL
LIN {X 0,Y 136.264,Z 454.516,A -85,B 0,C 180,E1 -24641.974,E2 -24641.974} C_VEL
LIN {X 0,Y 136.444,Z 454.493,A -85,B 0,C 180,E1 -24648.138,E2 -24648.138} C_VEL
LIN {X 0,Y 136.551,Z 454.479,A -85,B 0,C 180,E1 -24651.118,E2 -24651.118} C_VEL
LIN {X 0,Y 137.135,Z 454.403,A -85,B 0,C 180,E1 -24660,E2 -24660} C_VEL
LIN {X 0,Y 136.6,Z 454.468,A -85,B 0,C 180,E1 -24668.88,E2 -24668.88} C_VEL
LIN {X 0,Y 136.491,Z 454.468,A -85,B 0,C 180,E1 -24671.955,E2 -24671.955} C_VEL
LIN {X 0,Y 136.243,Z 454.5,A -85,B 0,C 180,E1 -24678.03,E2 -24678.03} C_VEL
LIN {X 0,Y 136.198,Z 454.464,A -85,B 0,C 180,E1 -24681.75,E2 -24681.75} C_VEL
LIN {X 0,Y 136.117,Z 454.528,A -85,B 0,C 180,E1 -24688.63,E2 -24688.63} C_VEL
LIN {X 0,Y 136.08,Z 454.496,A -85,B 0,C 180,E1 -24694.619,E2 -24694.619} C_VEL
LIN {X 0,Y 136.047,Z 454.529,A -85,B 0,C 180,E1 -24696.793,E2 -24696.793} C_VEL
LIN {X 0,Y 136.868,Z 457.023,A -85,B 0,C 180,E1 -24697.806,E2 -24697.806} C_VEL
LIN {X 0,Y 138.965,Z 459.442,A -85,B 0,C 180,E1 -24699.57,E2 -24699.57} C_VEL
LIN {X 0,Y 142.224,Z 464.846,A -85,B 0,C 180,E1 -24702.559,E2 -24702.559} C_VEL
LIN {X 0,Y 146.061,Z 471.882,A -85,B 0,C 180,E1 -24706.2,E2 -24706.2} C_VEL
LIN {X 0,Y 149.646,Z 479.798,A -85,B 0,C 180,E1 -24709.971,E2 -24709.971} C_VEL
LIN {X 0,Y 152.42,Z 488.367,A -85,B 0,C 180,E1 -24713.794,E2 -24713.794} C_VEL
LIN {X 0,Y 154.05,Z 495.104,A -85,B 0,C 180,E1 -24716.808,E2 -24716.808} C_VEL
LIN {X 0,Y 155.046,Z 502.279,A -85,B 0,C 180,E1 -24720.092,E2 -24720.092} C_VEL
LIN {X 0,Y 151.615,Z 510.617,A -85,B 0,C 180,E1 -24723.132,E2 -24723.132} C_VEL
LIN {X 0,Y 147.851,Z 518.734,A -85,B 0,C 180,E1 -24726.912,E2 -24726.912} C_VEL
LIN {X 0,Y 145.118,Z 524.289,A -85,B 0,C 180,E1 -24730.184,E2 -24730.184} C_VEL
LIN {X 0,Y 142.428,Z 529.691,A -85,B 0,C 180,E1 -24734.253,E2 -24734.253} C_VEL
LIN {X 0,Y 140.238,Z 533.946,A -85,B 0,C 180,E1 -24738.437,E2 -24738.437} C_VEL
LIN {X 0,Y 138.931,Z 536.227,A -85,B 0,C 180,E1 -24741.272,E2 -24741.272} C_VEL
LIN {X 0,Y 138.064,Z 538.065,A -85,B 0,C 180,E1 -24744.157,E2 -24744.157} C_VEL
LIN {X 0,Y 137.447,Z 539.457,A -85,B 0,C 180,E1 -24747.07,E2 -24747.07} C_VEL
LIN {X 0,Y 137.234,Z 541.046,A -85,B 0,C 180,E1 -24752.936,E2 -24752.936} C_VEL
LIN {X 0,Y 137.339,Z 541.311,A -85,B 0,C 180,E1 -24755.875,E2 -24755.875} C_VEL
LIN {X 0,Y 137.655,Z 541.17,A -85,B 0,C 180,E1 -24758.811,E2 -24758.811} C_VEL
LIN {X 0,Y 139.822,Z 539.634,A -85,B 0,C 180,E1 -24764.556,E2 -24764.556} C_VEL
LIN {X 0,Y 141.318,Z 538.293,A -85,B 0,C 180,E1 -24767.362,E2 -24767.362} C_VEL
LIN {X 0,Y 144.111,Z 535.031,A -85,B 0,C 180,E1 -24772.089,E2 -24772.089} C_VEL
LIN {X 0,Y 147.811,Z 530.178,A -85,B 0,C 180,E1 -24776.853,E2 -24776.853} C_VEL
LIN {X 0,Y 152.042,Z 523.872,A -85,B 0,C 180,E1 -24781.334,E2 -24781.334} C_VEL
LIN {X 0,Y 156.336,Z 516.882,A -85,B 0,C 180,E1 -24784.972,E2 -24784.972} C_VEL
LIN {X 0,Y 159.66,Z 510.672,A -85,B 0,C 180,E1 -24787.595,E2 -24787.595} C_VEL
LIN {X 0,Y 159.09,Z 503.678,A -85,B 0,C 180,E1 -24791.503,E2 -24791.503} C_VEL
LIN {X 0,Y 157.79,Z 496.381,A -85,B 0,C 180,E1 -24795.452,E2 -24795.452} C_VEL
LIN {X 0,Y 155.855,Z 489.659,A -85,B 0,C 180,E1 -24799.168,E2 -24799.168} C_VEL
LIN {X 0,Y 152.879,Z 481.767,A -85,B 0,C 180,E1 -24803.779,E2 -24803.779} C_VEL
LIN {X 0,Y 149.783,Z 475.097,A -85,B 0,C 180,E1 -24808.069,E2 -24808.069} C_VEL
LIN {X 0,Y 147.164,Z 470.618,A -85,B 0,C 180,E1 -24811.473,E2 -24811.473} C_VEL
LIN {X 0,Y 145.106,Z 467.668,A -85,B 0,C 180,E1 -24814.157,E2 -24814.157} C_VEL
LIN {X 0,Y 144.06,Z 465.408,A -85,B 0,C 180,E1 -24815.847,E2 -24815.847} C_VEL
LIN {X 0,Y 141.744,Z 463.073,A -85,B 0,C 180,E1 -24818.983,E2 -24818.983} C_VEL
LIN {X 0,Y 140.219,Z 465.033,A -85,B 0,C 180,E1 -24820.034,E2 -24820.034} C_VEL
LIN {X 0,Y 139.359,Z 465.595,A -85,B 0,C 180,E1 -24820.864,E2 -24820.864} C_VEL
LIN {X 0,Y 138.749,Z 465.137,A -85,B 0,C 180,E1 -24821.83,E2 -24821.83} C_VEL
LIN {X 0,Y 138.665,Z 464.389,A -85,B 0,C 180,E1 -24822.248,E2 -24822.248} C_VEL
LIN {X 0,Y 139.299,Z 466.79,A -85,B 0,C 180,E1 -24822.758,E2 -24822.758} C_VEL
LIN {X 0,Y 138.292,Z 478.383,A -85,B 0,C 180,E1 -24825.676,E2 -24825.676} C_VEL
LIN {X 0,Y 137.155,Z 490.233,A -85,B 0,C 180,E1 -24829.295,E2 -24829.295} C_VEL
LIN {X 0,Y 136.454,Z 499.32,A -85,B 0,C 180,E1 -24832.601,E2 -24832.601} C_VEL
LIN {X 0,Y 135.968,Z 509.579,A -85,B 0,C 180,E1 -24837.037,E2 -24837.037} C_VEL
LIN {X 0,Y 136.409,Z 519.666,A -85,B 0,C 180,E1 -24842.214,E2 -24842.214} C_VEL
LIN {X 0,Y 137.499,Z 527.95,A -85,B 0,C 180,E1 -24847.341,E2 -24847.341} C_VEL
LIN {X 0,Y 140.068,Z 535.764,A -85,B 0,C 180,E1 -24853.049,E2 -24853.049} C_VEL
LIN {X 0,Y 144.266,Z 542.112,A -85,B 0,C 180,E1 -24858.46,E2 -24858.46} C_VEL
LIN {X 0,Y 149.759,Z 547.01,A -85,B 0,C 180,E1 -24863.509,E2 -24863.509} C_VEL
LIN {X 0,Y 154.701,Z 549.895,A -85,B 0,C 180,E1 -24867.019,E2 -24867.019} C_VEL
LIN {X 0,Y 162.274,Z 552.618,A -85,B 0,C 180,E1 -24871.313,E2 -24871.313} C_VEL
LIN {X 0,Y 170.858,Z 554.138,A -85,B 0,C 180,E1 -24875.16,E2 -24875.16} C_VEL
LIN {X 0,Y 180.384,Z 554.47,A -85,B 0,C 180,E1 -24878.563,E2 -24878.563} C_VEL
LIN {X 0,Y 182.431,Z 554.629,A -85,B 0,C 180,E1 -24879.602,E2 -24879.602} C_VEL
LIN {X 0,Y 173.418,Z 558.581,A -85,B 0,C 180,E1 -24883.547,E2 -24883.547} C_VEL
LIN {X 0,Y 165.279,Z 561.518,A -85,B 0,C 180,E1 -24887.128,E2 -24887.128} C_VEL
LIN {X 0,Y 157.327,Z 563.854,A -85,B 0,C 180,E1 -24891.288,E2 -24891.288} C_VEL
LIN {X 0,Y 150.354,Z 565.35,A -85,B 0,C 180,E1 -24895.88,E2 -24895.88} C_VEL
LIN {X 0,Y 143.06,Z 565.932,A -85,B 0,C 180,E1 -24902.579,E2 -24902.579} C_VEL
LIN {X 0,Y 142.234,Z 565.954,A -85,B 0,C 180,E1 -24903.595,E2 -24903.595} C_VEL
LIN {X 0,Y 138.784,Z 570.792,A -85,B 0,C 180,E1 -24907.678,E2 -24907.678} C_VEL
LIN {X 0,Y 136.498,Z 574.593,A -85,B 0,C 180,E1 -24912.005,E2 -24912.005} C_VEL
LIN {X 0,Y 135.567,Z 576.611,A -85,B 0,C 180,E1 -24914.976,E2 -24914.976} C_VEL
LIN {X 0,Y 134.954,Z 579.354,A -85,B 0,C 180,E1 -24921.011,E2 -24921.011} C_VEL
LIN {X 0,Y 135.251,Z 580.151,A -85,B 0,C 180,E1 -24924.034,E2 -24924.034} C_VEL
LIN {X 0,Y 135.729,Z 580.536,A -85,B 0,C 180,E1 -24927.031,E2 -24927.031} C_VEL
LIN {X 0,Y 136.457,Z 580.475,A -85,B 0,C 180,E1 -24929.999,E2 -24929.999} C_VEL
LIN {X 0,Y 135.743,Z 579.762,A -85,B 0,C 180,E1 -24932.967,E2 -24932.967} C_VEL
LIN {X 0,Y 135.038,Z 577.329,A -85,B 0,C 180,E1 -24938.567,E2 -24938.567} C_VEL
LIN {X 0,Y 135.196,Z 573.916,A -85,B 0,C 180,E1 -24943.528,E2 -24943.528} C_VEL
LIN {X 0,Y 136.184,Z 569.682,A -85,B 0,C 180,E1 -24948.037,E2 -24948.037} C_VEL
LIN {X 0,Y 138.657,Z 563.295,A -85,B 0,C 180,E1 -24953.129,E2 -24953.129} C_VEL
LIN {X 0,Y 141.588,Z 556.37,A -85,B 0,C 180,E1 -24957.331,E2 -24957.331} C_VEL
LIN {X 0,Y 144.167,Z 547.613,A -85,B 0,C 180,E1 -24961.604,E2 -24961.604} C_VEL
LIN {X 0,Y 146.534,Z 538.583,A -85,B 0,C 180,E1 -24965.137,E2 -24965.137} C_VEL
LIN {X 0,Y 148.569,Z 528.619,A -85,B 0,C 180,E1 -24968.379,E2 -24968.379} C_VEL
LIN {X 0,Y 150.029,Z 517.569,A -85,B 0,C 180,E1 -24971.453,E2 -24971.453} C_VEL
LIN {X 0,Y 150.833,Z 505.531,A -85,B 0,C 180,E1 -24974.34,E2 -24974.34} C_VEL
LIN {X 0,Y 150.625,Z 494.477,A -85,B 0,C 180,E1 -24976.75,E2 -24976.75} C_VEL
LIN {X 0,Y 150.292,Z 492.101,A -85,B 0,C 180,E1 -24977.308,E2 -24977.308} C_VEL
LIN {X 0,Y 146.672,Z 482.475,A -85,B 0,C 180,E1 -24980.329,E2 -24980.329} C_VEL
LIN {X 0,Y 144.294,Z 476.996,A -85,B 0,C 180,E1 -24982.165,E2 -24982.165} C_VEL
LIN {X 0,Y 142.23,Z 472.663,A -85,B 0,C 180,E1 -24983.721,E2 -24983.721} C_VEL
LIN {X 0,Y 141.515,Z 470.992,A -85,B 0,C 180,E1 -24984.283,E2 -24984.283} C_VEL
LIN {X 0,Y 141.375,Z 470.818,A -85,B 0,C 180,E1 -24984.375,E2 -24984.375} C_VEL
LIN {X 0,Y 139.503,Z 468.904,A -85,B 0,C 180,E1 -24985.6,E2 -24985.6} C_VEL
LIN {X 0,Y 132.387,Z 465.738,A -85,B 0,C 180,E1 -24990.29,E2 -24990.29} C_VEL
LIN {X 0,Y 130.923,Z 463.575,A -85,B 0,C 180,E1 -24991.576,E2 -24991.576} C_VEL
LIN {X 0,Y 130.673,Z 462.67,A -85,B 0,C 180,E1 -24991.927,E2 -24991.927} C_VEL
LIN {X 0,Y 129.898,Z 458.952,A -85,B 0,C 180,E1 -24997.746,E2 -24997.746} C_VEL
LIN {X 0,Y 129.329,Z 456.15,A -85,B 0,C 180,E1 -25002.61,E2 -25002.61} C_VEL
LIN {X 0,Y 129.204,Z 455.395,A -85,B 0,C 180,E1 -25004.219,E2 -25004.219} C_VEL
LIN {X 0,Y 129.367,Z 455.374,A -85,B 0,C 180,E1 -25007.922,E2 -25007.922} C_VEL
LIN {X 0,Y 129.477,Z 455.36,A -85,B 0,C 180,E1 -25010.629,E2 -25010.629} C_VEL
LIN {X 0,Y 130.09,Z 455.28,A -85,B 0,C 180,E1 -25020,E2 -25020} C_VEL
LIN {X 0,Y 129.524,Z 455.35,A -85,B 0,C 180,E1 -25029.369,E2 -25029.369} C_VEL
LIN {X 0,Y 129.393,Z 455.35,A -85,B 0,C 180,E1 -25032.549,E2 -25032.549} C_VEL
LIN {X 0,Y 129.154,Z 455.364,A -85,B 0,C 180,E1 -25039.057,E2 -25039.057} C_VEL
LIN {X 0,Y 129.109,Z 455.345,A -85,B 0,C 180,E1 -25042.399,E2 -25042.399} C_VEL
LIN {X 0,Y 129.036,Z 455.402,A -85,B 0,C 180,E1 -25049.374,E2 -25049.374} C_VEL
LIN {X 0,Y 129,Z 455.394,A -85,B 0,C 180,E1 -25051.855,E2 -25051.855} C_VEL
LIN {X 0,Y 129.779,Z 457.835,A -85,B 0,C 180,E1 -25053.027,E2 -25053.027} C_VEL
LIN {X 0,Y 132.157,Z 460.438,A -85,B 0,C 180,E1 -25055.455,E2 -25055.455} C_VEL
